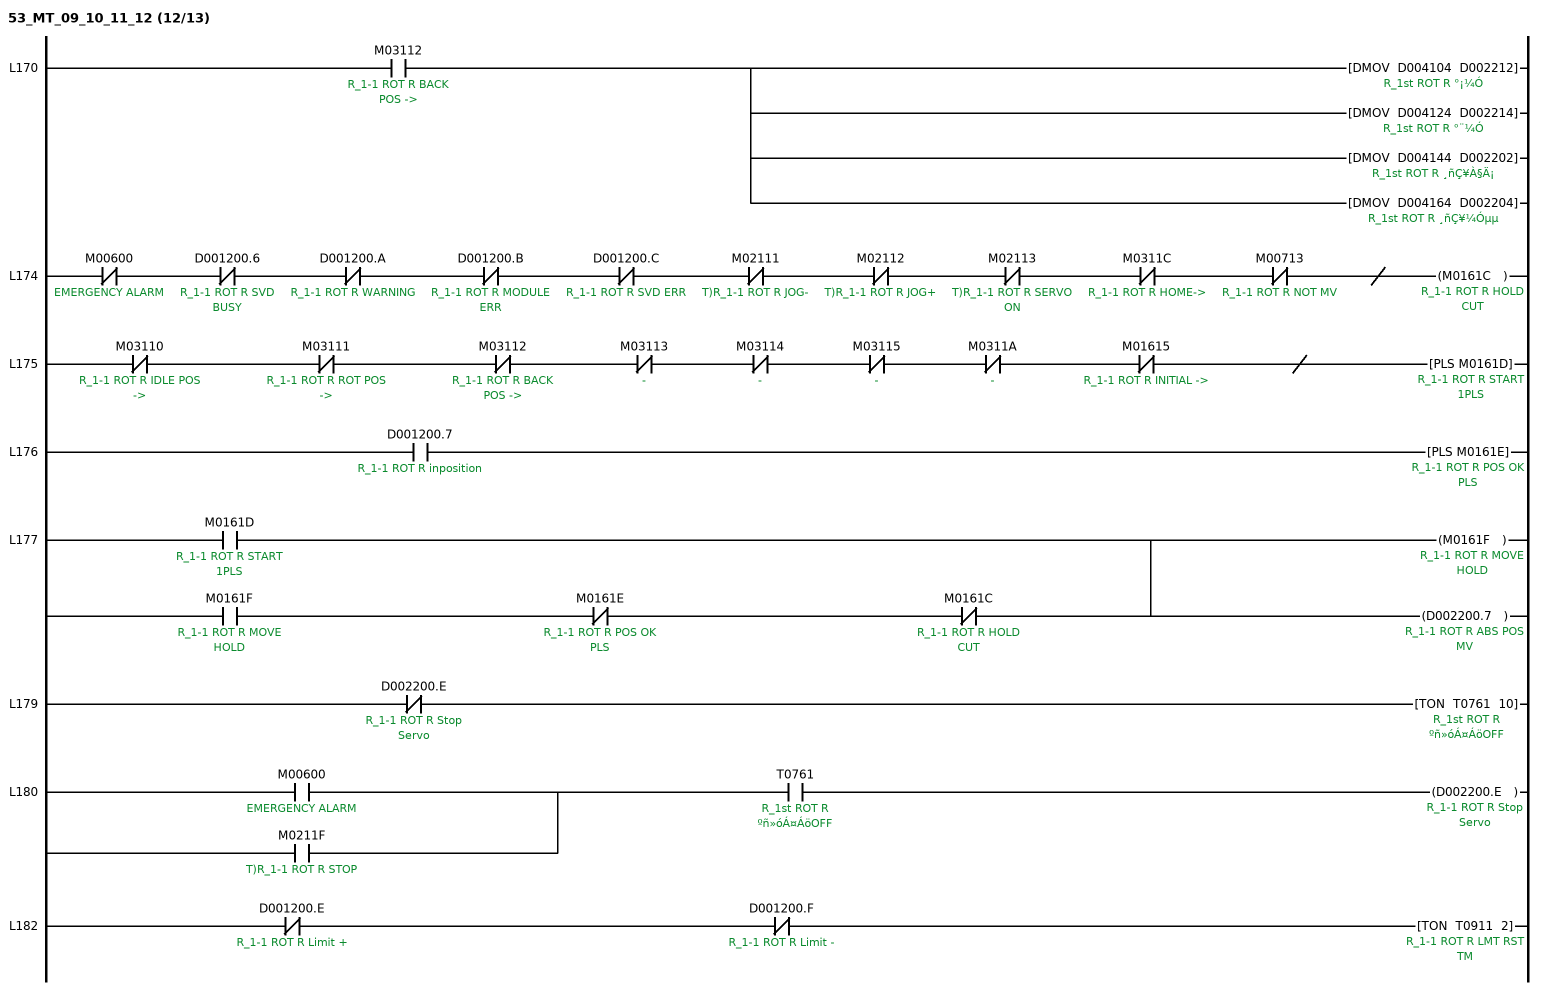
[picture p288: 53_MT_09_10_11_12 rungs L170-L182]
; L170
LOAD      M03112	// R_1-1 ROT R BACK POS ->
DMOV      D004104 D002212	// R_1st ROT R °¡¼Ó
DMOV      D004124 D002214	// R_1st ROT R °¨¼Ó
DMOV      D004144 D002202	// R_1st ROT R ¸ñÇ¥À§Ä¡
DMOV      D004164 D002204	// R_1st ROT R ¸ñÇ¥¼Óµµ
; L174
LOAD NOT  M00600	// EMERGENCY ALARM
AND NOT   D001200.6	// R_1-1 ROT R SVD BUSY
AND NOT   D001200.A	// R_1-1 ROT R WARNING
AND NOT   D001200.B	// R_1-1 ROT R MODULE ERR
AND NOT   D001200.C	// R_1-1 ROT R SVD ERR
AND NOT   M02111	// T)R_1-1 ROT R JOG-
AND NOT   M02112	// T)R_1-1 ROT R JOG+
AND NOT   M02113	// T)R_1-1 ROT R SERVO ON
AND NOT   M0311C	// R_1-1 ROT R HOME->
AND NOT   M00713	// R_1-1 ROT R NOT MV
NOT
OUT       M0161C	// R_1-1 ROT R HOLD CUT
; L175
LOAD NOT  M03110	// R_1-1 ROT R IDLE POS ->
AND NOT   M03111	// R_1-1 ROT R ROT POS ->
AND NOT   M03112	// R_1-1 ROT R BACK POS ->
AND NOT   M03113	// -
AND NOT   M03114	// -
AND NOT   M03115	// -
AND NOT   M0311A	// -
AND NOT   M01615	// R_1-1 ROT R INITIAL ->
NOT
OUTP      M0161D	// R_1-1 ROT R START 1PLS
; L176
LOAD      D001200.7	// R_1-1 ROT R inposition
OUTP      M0161E	// R_1-1 ROT R POS OK PLS
; L177
LOAD      M0161D	// R_1-1 ROT R START 1PLS
LOAD      M0161F	// R_1-1 ROT R MOVE HOLD
AND NOT   M0161E	// R_1-1 ROT R POS OK PLS
AND NOT   M0161C	// R_1-1 ROT R HOLD CUT
OR LOAD
OUT       M0161F	// R_1-1 ROT R MOVE HOLD
OUT       D002200.7	// R_1-1 ROT R ABS POS MV
; L179
LOAD NOT  D002200.E	// R_1-1 ROT R Stop Servo
TON       T0761 10	// R_1st ROT R ºñ»óÁ¤ÁöOFF
; L180
LOAD      M00600	// EMERGENCY ALARM
OR        M0211F	// T)R_1-1 ROT R STOP
AND       T0761	// R_1st ROT R ºñ»óÁ¤ÁöOFF
OUT       D002200.E	// R_1-1 ROT R Stop Servo
; L182
LOAD NOT  D001200.E	// R_1-1 ROT R Limit +
AND NOT   D001200.F	// R_1-1 ROT R Limit -
TON       T0911 2	// R_1-1 ROT R LMT RST TM

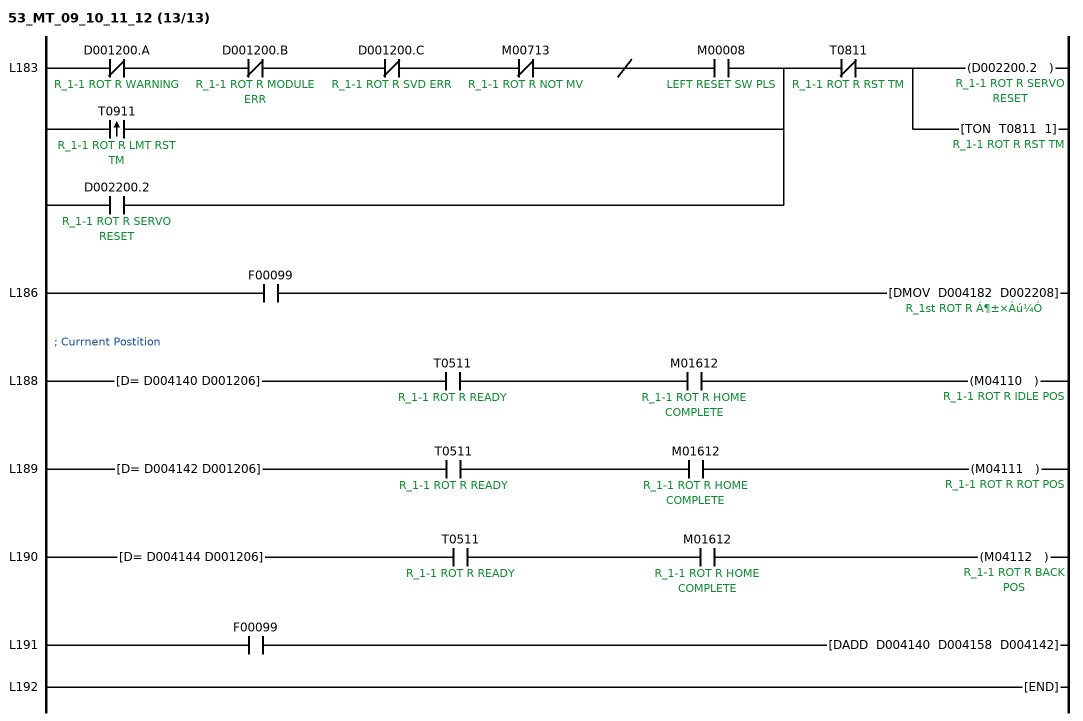
; L183
LOAD NOT  D001200.A	// R_1-1 ROT R WARNING
AND NOT   D001200.B	// R_1-1 ROT R MODULE ERR
AND NOT   D001200.C	// R_1-1 ROT R SVD ERR
AND NOT   M00713	// R_1-1 ROT R NOT MV
NOT
AND       M00008	// LEFT RESET SW PLS
ORP       T0911	// R_1-1 ROT R LMT RST TM
OR        D002200.2	// R_1-1 ROT R SERVO RESET
AND NOT   T0811	// R_1-1 ROT R RST TM
OUT       D002200.2	// R_1-1 ROT R SERVO RESET
TON       T0811 1	// R_1-1 ROT R RST TM
; L186
LOAD      F00099
DMOV      D004182 D002208	// R_1st ROT R Á¶±×Àú¼Ó
// Currnent Postition
; L188
LOADD=    D004140 D001206
AND       T0511	// R_1-1 ROT R READY
AND       M01612	// R_1-1 ROT R HOME COMPLETE
OUT       M04110	// R_1-1 ROT R IDLE POS
; L189
LOADD=    D004142 D001206
AND       T0511	// R_1-1 ROT R READY
AND       M01612	// R_1-1 ROT R HOME COMPLETE
OUT       M04111	// R_1-1 ROT R ROT POS
; L190
LOADD=    D004144 D001206
AND       T0511	// R_1-1 ROT R READY
AND       M01612	// R_1-1 ROT R HOME COMPLETE
OUT       M04112	// R_1-1 ROT R BACK POS
; L191
LOAD      F00099
DADD      D004140 D004158 D004142
; L192
END

PROGRAM 54_MT_13_14_15_16 (task: ½ºÄµ ÇÁ·Î±×·¥)

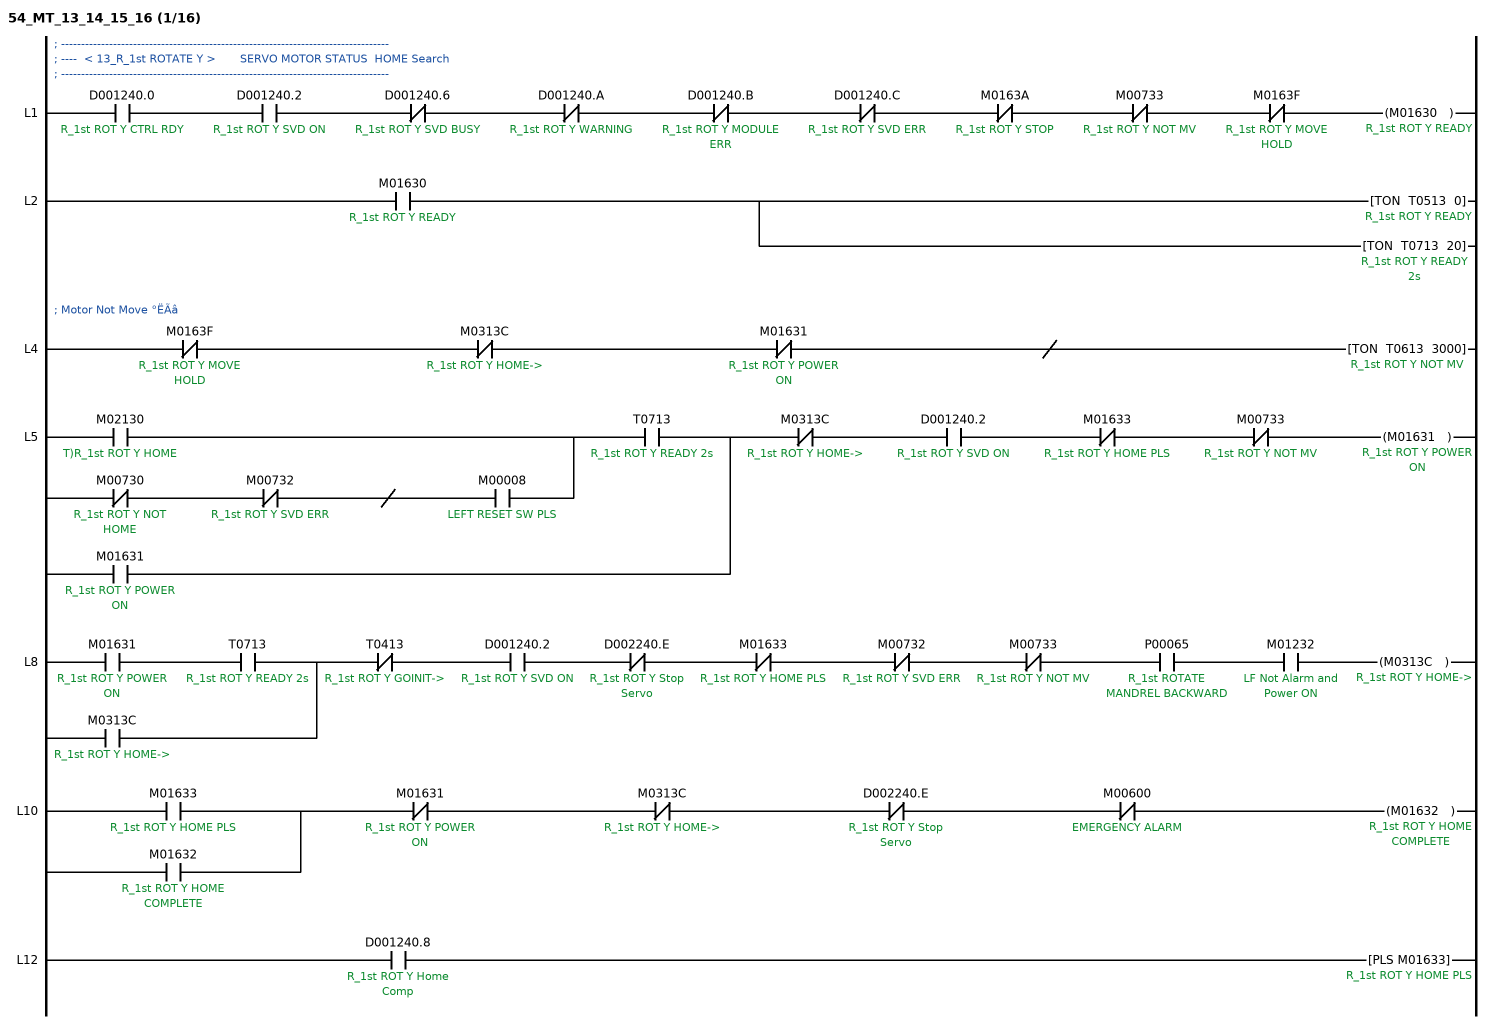
// ----------------------------------------------------------------------------------
// 
// ----  < 13_R_1st ROTATE Y >       SERVO MOTOR STATUS  HOME Search
// 
// ----------------------------------------------------------------------------------
; L1
LOAD      D001240.0	// R_1st ROT Y CTRL RDY
AND       D001240.2	// R_1st ROT Y SVD ON
AND NOT   D001240.6	// R_1st ROT Y SVD BUSY
AND NOT   D001240.A	// R_1st ROT Y WARNING
AND NOT   D001240.B	// R_1st ROT Y MODULE ERR
AND NOT   D001240.C	// R_1st ROT Y SVD ERR
AND NOT   M0163A	// R_1st ROT Y STOP
AND NOT   M00733	// R_1st ROT Y NOT MV
AND NOT   M0163F	// R_1st ROT Y MOVE HOLD
OUT       M01630	// R_1st ROT Y READY
; L2
LOAD      M01630	// R_1st ROT Y READY
TON       T0513 0	// R_1st ROT Y READY
TON       T0713 20	// R_1st ROT Y READY 2s
; L4
LOAD NOT  M0163F	// R_1st ROT Y MOVE HOLD
AND NOT   M0313C	// R_1st ROT Y HOME->
AND NOT   M01631	// R_1st ROT Y POWER ON
NOT
TON       T0613 3000	// R_1st ROT Y NOT MV
// output comment: Motor Not Move °ËÃâ
; L5
LOAD      M02130	// T)R_1st ROT Y HOME
LOAD NOT  M00730	// R_1st ROT Y NOT HOME
AND NOT   M00732	// R_1st ROT Y SVD ERR
NOT
AND       M00008	// LEFT RESET SW PLS
OR LOAD
AND       T0713	// R_1st ROT Y READY 2s
OR        M01631	// R_1st ROT Y POWER ON
AND NOT   M0313C	// R_1st ROT Y HOME->
AND       D001240.2	// R_1st ROT Y SVD ON
AND NOT   M01633	// R_1st ROT Y HOME PLS
AND NOT   M00733	// R_1st ROT Y NOT MV
OUT       M01631	// R_1st ROT Y POWER ON
; L8
LOAD      M01631	// R_1st ROT Y POWER ON
AND       T0713	// R_1st ROT Y READY 2s
OR        M0313C	// R_1st ROT Y HOME->
AND NOT   T0413	// R_1st ROT Y GOINIT->
AND       D001240.2	// R_1st ROT Y SVD ON
AND NOT   D002240.E	// R_1st ROT Y Stop Servo
AND NOT   M01633	// R_1st ROT Y HOME PLS
AND NOT   M00732	// R_1st ROT Y SVD ERR
AND NOT   M00733	// R_1st ROT Y NOT MV
AND       P00065	// R_1st ROTATE MANDREL BACKWARD
AND       M01232	// LF Not Alarm and Power ON
OUT       M0313C	// R_1st ROT Y HOME->
; L10
LOAD      M01633	// R_1st ROT Y HOME PLS
OR        M01632	// R_1st ROT Y HOME COMPLETE
AND NOT   M01631	// R_1st ROT Y POWER ON
AND NOT   M0313C	// R_1st ROT Y HOME->
AND NOT   D002240.E	// R_1st ROT Y Stop Servo
AND NOT   M00600	// EMERGENCY ALARM
OUT       M01632	// R_1st ROT Y HOME COMPLETE
; L12
LOAD      D001240.8	// R_1st ROT Y Home Comp
OUTP      M01633	// R_1st ROT Y HOME PLS

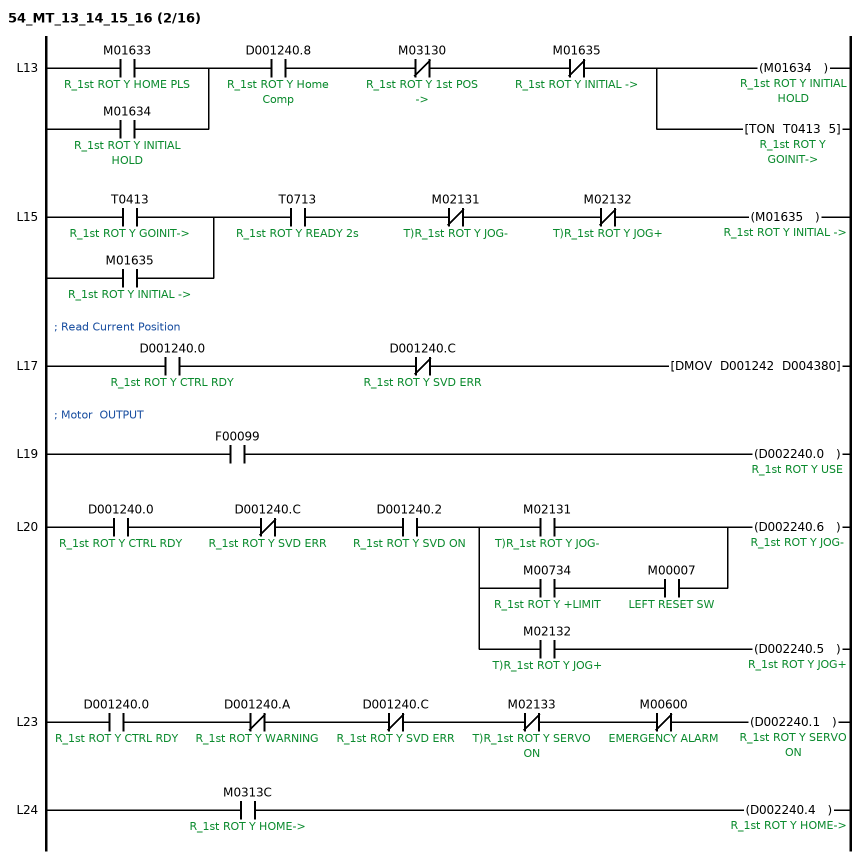
; L13
LOAD      M01633	// R_1st ROT Y HOME PLS
OR        M01634	// R_1st ROT Y INITIAL HOLD
AND       D001240.8	// R_1st ROT Y Home Comp
AND NOT   M03130	// R_1st ROT Y 1st POS ->
AND NOT   M01635	// R_1st ROT Y INITIAL ->
OUT       M01634	// R_1st ROT Y INITIAL HOLD
TON       T0413 5	// R_1st ROT Y GOINIT->
; L15
LOAD      T0413	// R_1st ROT Y GOINIT->
OR        M01635	// R_1st ROT Y INITIAL ->
AND       T0713	// R_1st ROT Y READY 2s
AND NOT   M02131	// T)R_1st ROT Y JOG-
AND NOT   M02132	// T)R_1st ROT Y JOG+
OUT       M01635	// R_1st ROT Y INITIAL ->
; L17
LOAD      D001240.0	// R_1st ROT Y CTRL RDY
AND NOT   D001240.C	// R_1st ROT Y SVD ERR
DMOV      D001242 D004380
// output comment: Read Current Position
//  Motor  OUTPUT
; L19
LOAD      F00099
OUT       D002240.0	// R_1st ROT Y USE
; L20
LOAD      D001240.0	// R_1st ROT Y CTRL RDY
AND NOT   D001240.C	// R_1st ROT Y SVD ERR
AND       D001240.2	// R_1st ROT Y SVD ON
MPUSH
LOAD      M02131	// T)R_1st ROT Y JOG-
LOAD      M00734	// R_1st ROT Y +LIMIT
AND       M00007	// LEFT RESET SW
OR LOAD
AND LOAD
OUT       D002240.6	// R_1st ROT Y JOG-
MPOP
AND       M02132	// T)R_1st ROT Y JOG+
OUT       D002240.5	// R_1st ROT Y JOG+
; L23
LOAD      D001240.0	// R_1st ROT Y CTRL RDY
AND NOT   D001240.A	// R_1st ROT Y WARNING
AND NOT   D001240.C	// R_1st ROT Y SVD ERR
AND NOT   M02133	// T)R_1st ROT Y SERVO ON
AND NOT   M00600	// EMERGENCY ALARM
OUT       D002240.1	// R_1st ROT Y SERVO ON
; L24
LOAD      M0313C	// R_1st ROT Y HOME->
OUT       D002240.4	// R_1st ROT Y HOME->

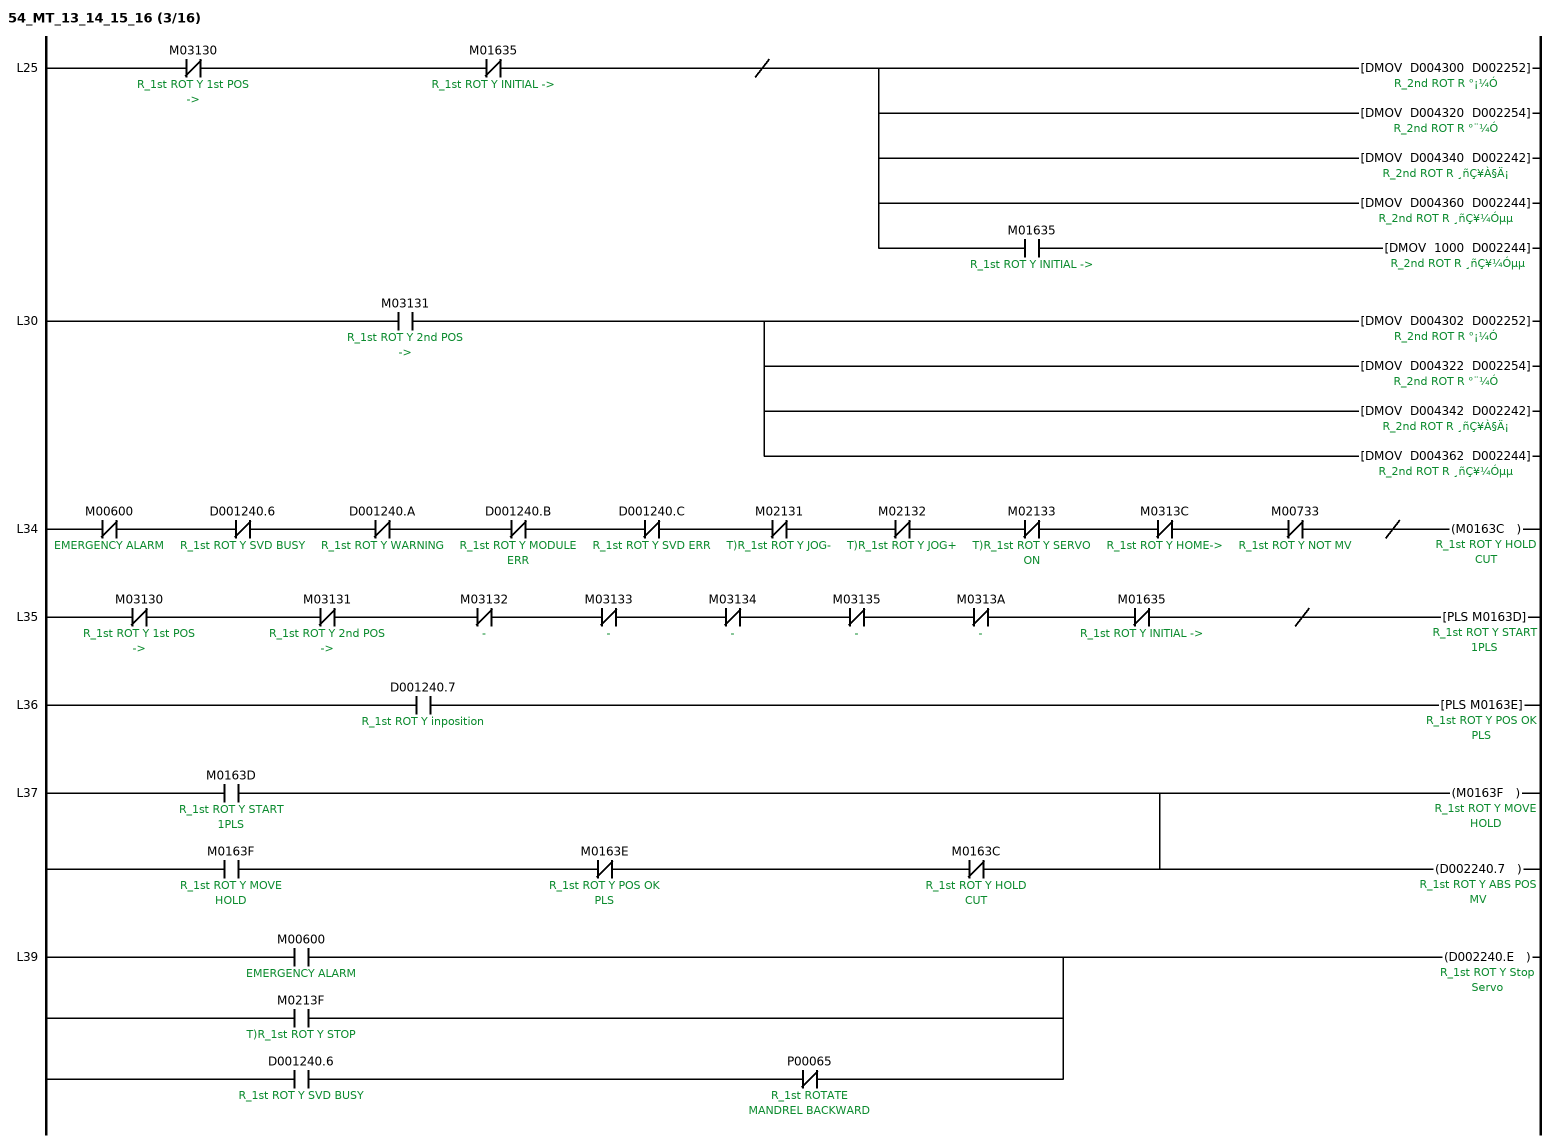
; L25
LOAD NOT  M03130	// R_1st ROT Y 1st POS ->
AND NOT   M01635	// R_1st ROT Y INITIAL ->
NOT
DMOV      D004300 D002252	// R_2nd ROT R °¡¼Ó
DMOV      D004320 D002254	// R_2nd ROT R °¨¼Ó
DMOV      D004340 D002242	// R_2nd ROT R ¸ñÇ¥À§Ä¡
DMOV      D004360 D002244	// R_2nd ROT R ¸ñÇ¥¼Óµµ
AND       M01635	// R_1st ROT Y INITIAL ->
DMOV      1000 D002244	// R_2nd ROT R ¸ñÇ¥¼Óµµ
; L30
LOAD      M03131	// R_1st ROT Y 2nd POS ->
DMOV      D004302 D002252	// R_2nd ROT R °¡¼Ó
DMOV      D004322 D002254	// R_2nd ROT R °¨¼Ó
DMOV      D004342 D002242	// R_2nd ROT R ¸ñÇ¥À§Ä¡
DMOV      D004362 D002244	// R_2nd ROT R ¸ñÇ¥¼Óµµ
; L34
LOAD NOT  M00600	// EMERGENCY ALARM
AND NOT   D001240.6	// R_1st ROT Y SVD BUSY
AND NOT   D001240.A	// R_1st ROT Y WARNING
AND NOT   D001240.B	// R_1st ROT Y MODULE ERR
AND NOT   D001240.C	// R_1st ROT Y SVD ERR
AND NOT   M02131	// T)R_1st ROT Y JOG-
AND NOT   M02132	// T)R_1st ROT Y JOG+
AND NOT   M02133	// T)R_1st ROT Y SERVO ON
AND NOT   M0313C	// R_1st ROT Y HOME->
AND NOT   M00733	// R_1st ROT Y NOT MV
NOT
OUT       M0163C	// R_1st ROT Y HOLD CUT
; L35
LOAD NOT  M03130	// R_1st ROT Y 1st POS ->
AND NOT   M03131	// R_1st ROT Y 2nd POS ->
AND NOT   M03132	// -
AND NOT   M03133	// -
AND NOT   M03134	// -
AND NOT   M03135	// -
AND NOT   M0313A	// -
AND NOT   M01635	// R_1st ROT Y INITIAL ->
NOT
OUTP      M0163D	// R_1st ROT Y START 1PLS
; L36
LOAD      D001240.7	// R_1st ROT Y inposition
OUTP      M0163E	// R_1st ROT Y POS OK PLS
; L37
LOAD      M0163D	// R_1st ROT Y START 1PLS
LOAD      M0163F	// R_1st ROT Y MOVE HOLD
AND NOT   M0163E	// R_1st ROT Y POS OK PLS
AND NOT   M0163C	// R_1st ROT Y HOLD CUT
OR LOAD
OUT       M0163F	// R_1st ROT Y MOVE HOLD
OUT       D002240.7	// R_1st ROT Y ABS POS MV
; L39
LOAD      M00600	// EMERGENCY ALARM
OR        M0213F	// T)R_1st ROT Y STOP
LOAD      D001240.6	// R_1st ROT Y SVD BUSY
AND NOT   P00065	// R_1st ROTATE MANDREL BACKWARD
OR LOAD
OUT       D002240.E	// R_1st ROT Y Stop Servo

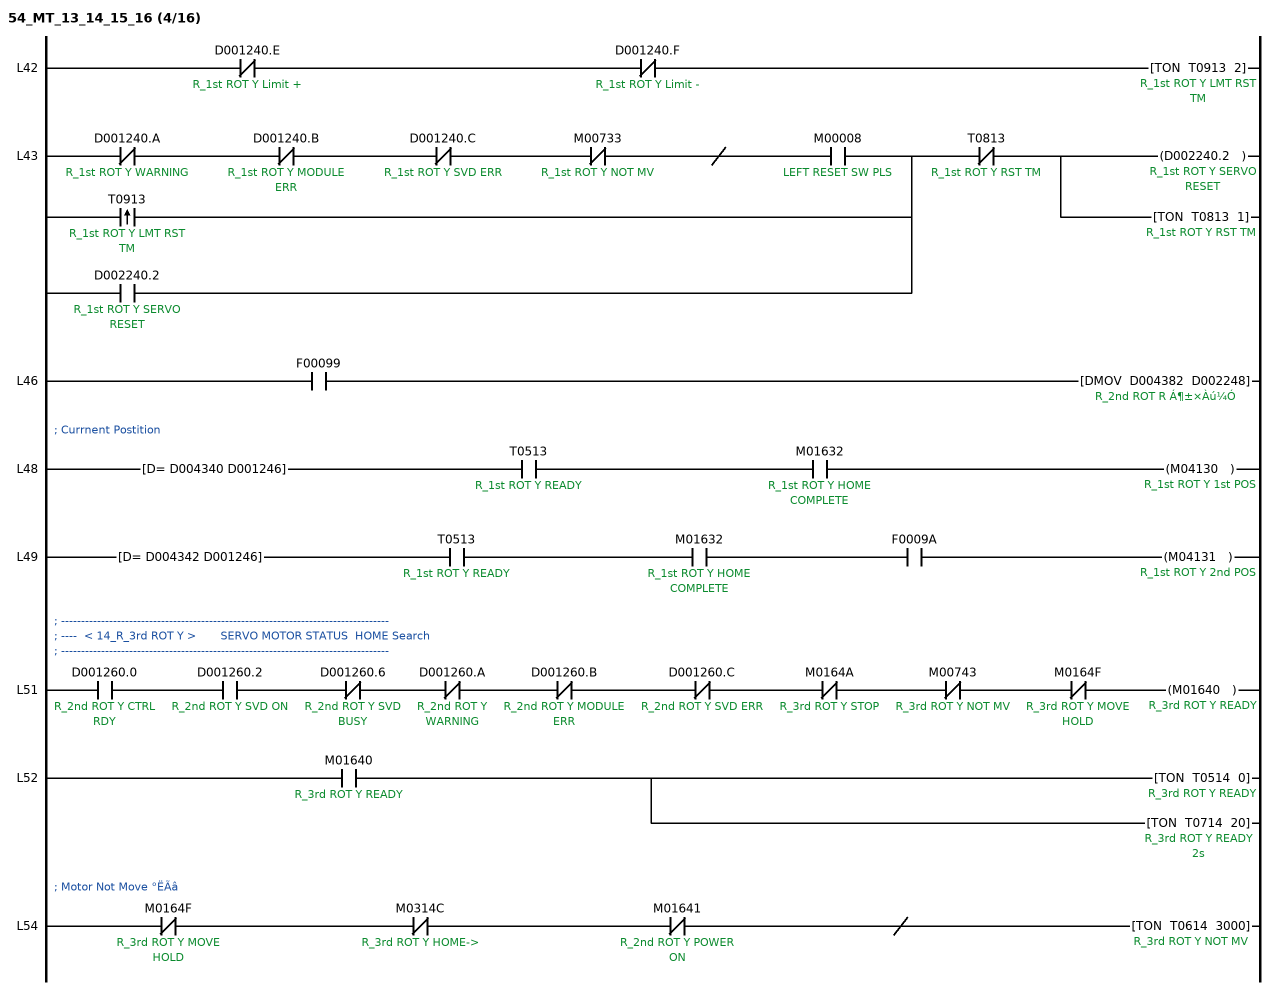
; L42
LOAD NOT  D001240.E	// R_1st ROT Y Limit +
AND NOT   D001240.F	// R_1st ROT Y Limit -
TON       T0913 2	// R_1st ROT Y LMT RST TM
; L43
LOAD NOT  D001240.A	// R_1st ROT Y WARNING
AND NOT   D001240.B	// R_1st ROT Y MODULE ERR
AND NOT   D001240.C	// R_1st ROT Y SVD ERR
AND NOT   M00733	// R_1st ROT Y NOT MV
NOT
AND       M00008	// LEFT RESET SW PLS
ORP       T0913	// R_1st ROT Y LMT RST TM
OR        D002240.2	// R_1st ROT Y SERVO RESET
AND NOT   T0813	// R_1st ROT Y RST TM
OUT       D002240.2	// R_1st ROT Y SERVO RESET
TON       T0813 1	// R_1st ROT Y RST TM
; L46
LOAD      F00099
DMOV      D004382 D002248	// R_2nd ROT R Á¶±×Àú¼Ó
// Currnent Postition
; L48
LOADD=    D004340 D001246
AND       T0513	// R_1st ROT Y READY
AND       M01632	// R_1st ROT Y HOME COMPLETE
OUT       M04130	// R_1st ROT Y 1st POS
; L49
LOADD=    D004342 D001246
AND       T0513	// R_1st ROT Y READY
AND       M01632	// R_1st ROT Y HOME COMPLETE
AND       F0009A
OUT       M04131	// R_1st ROT Y 2nd POS
// ----------------------------------------------------------------------------------
// 
// ----  < 14_R_3rd ROT Y >       SERVO MOTOR STATUS  HOME Search
// 
// ----------------------------------------------------------------------------------
; L51
LOAD      D001260.0	// R_2nd ROT Y CTRL RDY
AND       D001260.2	// R_2nd ROT Y SVD ON
AND NOT   D001260.6	// R_2nd ROT Y SVD BUSY
AND NOT   D001260.A	// R_2nd ROT Y WARNING
AND NOT   D001260.B	// R_2nd ROT Y MODULE ERR
AND NOT   D001260.C	// R_2nd ROT Y SVD ERR
AND NOT   M0164A	// R_3rd ROT Y STOP
AND NOT   M00743	// R_3rd ROT Y NOT MV
AND NOT   M0164F	// R_3rd ROT Y MOVE HOLD
OUT       M01640	// R_3rd ROT Y READY
; L52
LOAD      M01640	// R_3rd ROT Y READY
TON       T0514 0	// R_3rd ROT Y READY
TON       T0714 20	// R_3rd ROT Y READY 2s
; L54
LOAD NOT  M0164F	// R_3rd ROT Y MOVE HOLD
AND NOT   M0314C	// R_3rd ROT Y HOME->
AND NOT   M01641	// R_2nd ROT Y POWER ON
NOT
TON       T0614 3000	// R_3rd ROT Y NOT MV
// output comment: Motor Not Move °ËÃâ

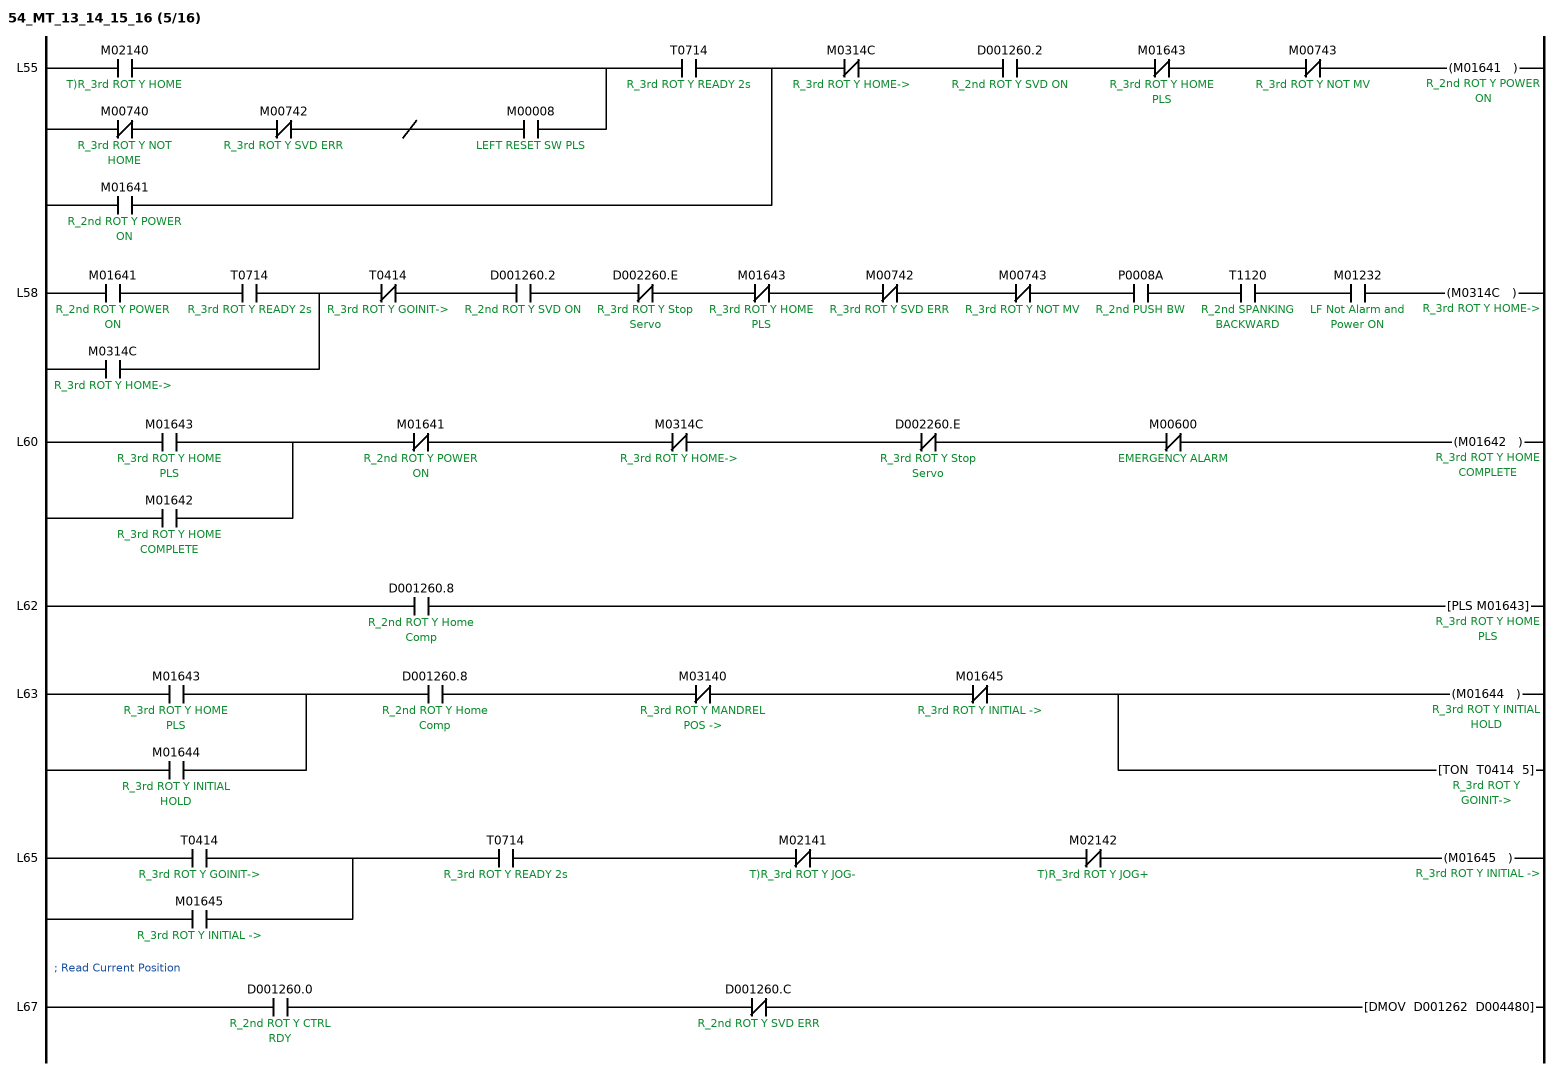
; L55
LOAD      M02140	// T)R_3rd ROT Y HOME
LOAD NOT  M00740	// R_3rd ROT Y NOT HOME
AND NOT   M00742	// R_3rd ROT Y SVD ERR
NOT
AND       M00008	// LEFT RESET SW PLS
OR LOAD
AND       T0714	// R_3rd ROT Y READY 2s
OR        M01641	// R_2nd ROT Y POWER ON
AND NOT   M0314C	// R_3rd ROT Y HOME->
AND       D001260.2	// R_2nd ROT Y SVD ON
AND NOT   M01643	// R_3rd ROT Y HOME PLS
AND NOT   M00743	// R_3rd ROT Y NOT MV
OUT       M01641	// R_2nd ROT Y POWER ON
; L58
LOAD      M01641	// R_2nd ROT Y POWER ON
AND       T0714	// R_3rd ROT Y READY 2s
OR        M0314C	// R_3rd ROT Y HOME->
AND NOT   T0414	// R_3rd ROT Y GOINIT->
AND       D001260.2	// R_2nd ROT Y SVD ON
AND NOT   D002260.E	// R_3rd ROT Y Stop Servo
AND NOT   M01643	// R_3rd ROT Y HOME PLS
AND NOT   M00742	// R_3rd ROT Y SVD ERR
AND NOT   M00743	// R_3rd ROT Y NOT MV
AND       P0008A	// R_2nd PUSH BW
AND       T1120	// R_2nd SPANKING BACKWARD
AND       M01232	// LF Not Alarm and Power ON
OUT       M0314C	// R_3rd ROT Y HOME->
; L60
LOAD      M01643	// R_3rd ROT Y HOME PLS
OR        M01642	// R_3rd ROT Y HOME COMPLETE
AND NOT   M01641	// R_2nd ROT Y POWER ON
AND NOT   M0314C	// R_3rd ROT Y HOME->
AND NOT   D002260.E	// R_3rd ROT Y Stop Servo
AND NOT   M00600	// EMERGENCY ALARM
OUT       M01642	// R_3rd ROT Y HOME COMPLETE
; L62
LOAD      D001260.8	// R_2nd ROT Y Home Comp
OUTP      M01643	// R_3rd ROT Y HOME PLS
; L63
LOAD      M01643	// R_3rd ROT Y HOME PLS
OR        M01644	// R_3rd ROT Y INITIAL HOLD
AND       D001260.8	// R_2nd ROT Y Home Comp
AND NOT   M03140	// R_3rd ROT Y MANDREL POS ->
AND NOT   M01645	// R_3rd ROT Y INITIAL ->
OUT       M01644	// R_3rd ROT Y INITIAL HOLD
TON       T0414 5	// R_3rd ROT Y GOINIT->
; L65
LOAD      T0414	// R_3rd ROT Y GOINIT->
OR        M01645	// R_3rd ROT Y INITIAL ->
AND       T0714	// R_3rd ROT Y READY 2s
AND NOT   M02141	// T)R_3rd ROT Y JOG-
AND NOT   M02142	// T)R_3rd ROT Y JOG+
OUT       M01645	// R_3rd ROT Y INITIAL ->
; L67
LOAD      D001260.0	// R_2nd ROT Y CTRL RDY
AND NOT   D001260.C	// R_2nd ROT Y SVD ERR
DMOV      D001262 D004480
// output comment: Read Current Position

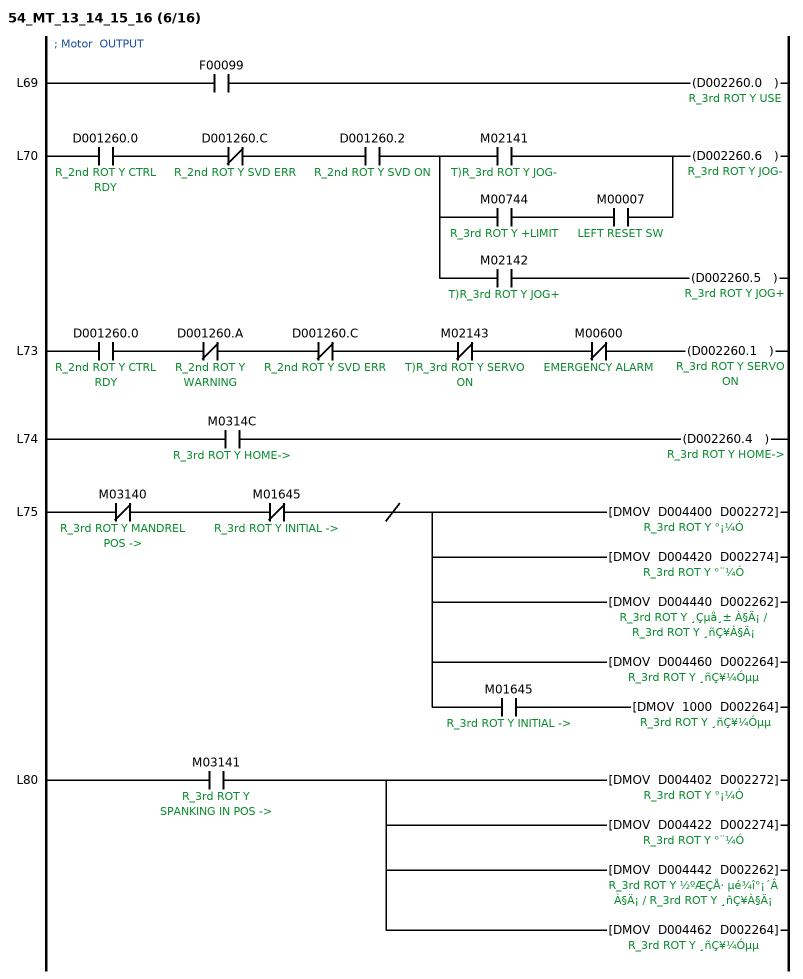
//  Motor  OUTPUT
; L69
LOAD      F00099
OUT       D002260.0	// R_3rd ROT Y USE
; L70
LOAD      D001260.0	// R_2nd ROT Y CTRL RDY
AND NOT   D001260.C	// R_2nd ROT Y SVD ERR
AND       D001260.2	// R_2nd ROT Y SVD ON
MPUSH
LOAD      M02141	// T)R_3rd ROT Y JOG-
LOAD      M00744	// R_3rd ROT Y +LIMIT
AND       M00007	// LEFT RESET SW
OR LOAD
AND LOAD
OUT       D002260.6	// R_3rd ROT Y JOG-
MPOP
AND       M02142	// T)R_3rd ROT Y JOG+
OUT       D002260.5	// R_3rd ROT Y JOG+
; L73
LOAD      D001260.0	// R_2nd ROT Y CTRL RDY
AND NOT   D001260.A	// R_2nd ROT Y WARNING
AND NOT   D001260.C	// R_2nd ROT Y SVD ERR
AND NOT   M02143	// T)R_3rd ROT Y SERVO ON
AND NOT   M00600	// EMERGENCY ALARM
OUT       D002260.1	// R_3rd ROT Y SERVO ON
; L74
LOAD      M0314C	// R_3rd ROT Y HOME->
OUT       D002260.4	// R_3rd ROT Y HOME->
; L75
LOAD NOT  M03140	// R_3rd ROT Y MANDREL POS ->
AND NOT   M01645	// R_3rd ROT Y INITIAL ->
NOT
DMOV      D004400 D002272	// R_3rd ROT Y °¡¼Ó
DMOV      D004420 D002274	// R_3rd ROT Y °¨¼Ó
DMOV      D004440 D002262	// R_3rd ROT Y ¸Çµå¸± À§Ä¡ / R_3rd ROT Y ¸ñÇ¥À§Ä¡
DMOV      D004460 D002264	// R_3rd ROT Y ¸ñÇ¥¼Óµµ
AND       M01645	// R_3rd ROT Y INITIAL ->
DMOV      1000 D002264	// R_3rd ROT Y ¸ñÇ¥¼Óµµ
; L80
LOAD      M03141	// R_3rd ROT Y SPANKING IN POS ->
DMOV      D004402 D002272	// R_3rd ROT Y °¡¼Ó
DMOV      D004422 D002274	// R_3rd ROT Y °¨¼Ó
DMOV      D004442 D002262	// R_3rd ROT Y ½ºÆÇÅ· µé¾î°¡´Â À§Ä¡ / R_3rd ROT Y ¸ñÇ¥À§Ä¡
DMOV      D004462 D002264	// R_3rd ROT Y ¸ñÇ¥¼Óµµ

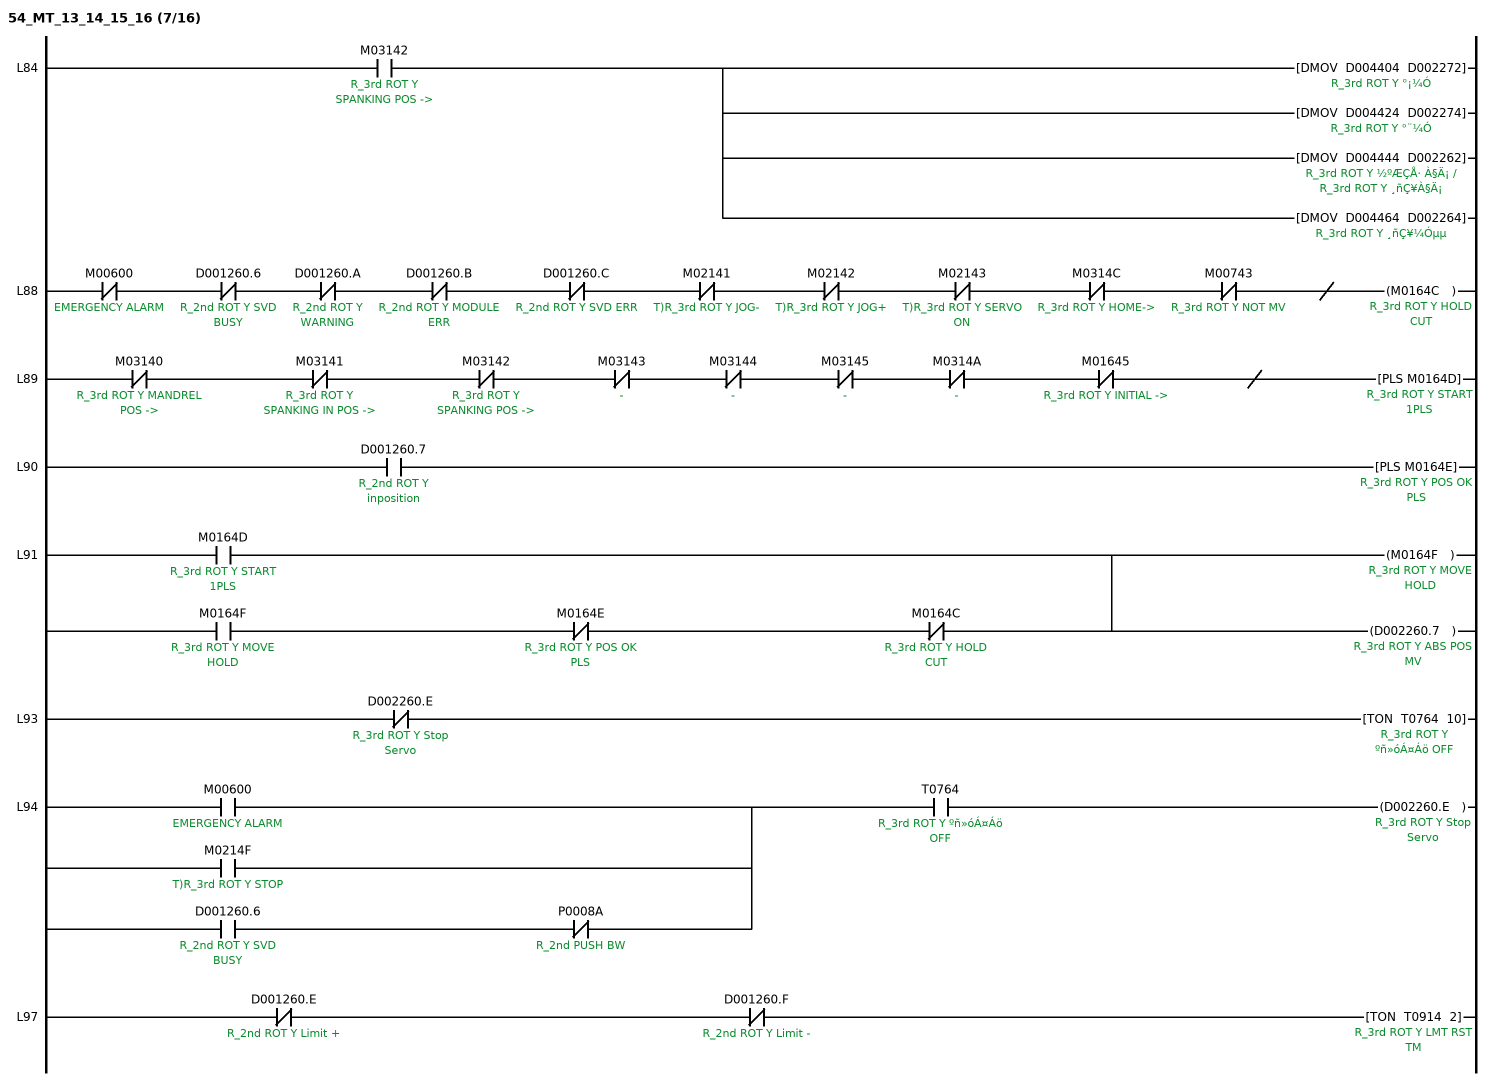
; L84
LOAD      M03142	// R_3rd ROT Y SPANKING POS ->
DMOV      D004404 D002272	// R_3rd ROT Y °¡¼Ó
DMOV      D004424 D002274	// R_3rd ROT Y °¨¼Ó
DMOV      D004444 D002262	// R_3rd ROT Y ½ºÆÇÅ· À§Ä¡ / R_3rd ROT Y ¸ñÇ¥À§Ä¡
DMOV      D004464 D002264	// R_3rd ROT Y ¸ñÇ¥¼Óµµ
; L88
LOAD NOT  M00600	// EMERGENCY ALARM
AND NOT   D001260.6	// R_2nd ROT Y SVD BUSY
AND NOT   D001260.A	// R_2nd ROT Y WARNING
AND NOT   D001260.B	// R_2nd ROT Y MODULE ERR
AND NOT   D001260.C	// R_2nd ROT Y SVD ERR
AND NOT   M02141	// T)R_3rd ROT Y JOG-
AND NOT   M02142	// T)R_3rd ROT Y JOG+
AND NOT   M02143	// T)R_3rd ROT Y SERVO ON
AND NOT   M0314C	// R_3rd ROT Y HOME->
AND NOT   M00743	// R_3rd ROT Y NOT MV
NOT
OUT       M0164C	// R_3rd ROT Y HOLD CUT
; L89
LOAD NOT  M03140	// R_3rd ROT Y MANDREL POS ->
AND NOT   M03141	// R_3rd ROT Y SPANKING IN POS ->
AND NOT   M03142	// R_3rd ROT Y SPANKING POS ->
AND NOT   M03143	// -
AND NOT   M03144	// -
AND NOT   M03145	// -
AND NOT   M0314A	// -
AND NOT   M01645	// R_3rd ROT Y INITIAL ->
NOT
OUTP      M0164D	// R_3rd ROT Y START 1PLS
; L90
LOAD      D001260.7	// R_2nd ROT Y inposition
OUTP      M0164E	// R_3rd ROT Y POS OK PLS
; L91
LOAD      M0164D	// R_3rd ROT Y START 1PLS
LOAD      M0164F	// R_3rd ROT Y MOVE HOLD
AND NOT   M0164E	// R_3rd ROT Y POS OK PLS
AND NOT   M0164C	// R_3rd ROT Y HOLD CUT
OR LOAD
OUT       M0164F	// R_3rd ROT Y MOVE HOLD
OUT       D002260.7	// R_3rd ROT Y ABS POS MV
; L93
LOAD NOT  D002260.E	// R_3rd ROT Y Stop Servo
TON       T0764 10	// R_3rd ROT Y ºñ»óÁ¤Áö OFF
; L94
LOAD      M00600	// EMERGENCY ALARM
OR        M0214F	// T)R_3rd ROT Y STOP
LOAD      D001260.6	// R_2nd ROT Y SVD BUSY
AND NOT   P0008A	// R_2nd PUSH BW
OR LOAD
AND       T0764	// R_3rd ROT Y ºñ»óÁ¤Áö OFF
OUT       D002260.E	// R_3rd ROT Y Stop Servo
; L97
LOAD NOT  D001260.E	// R_2nd ROT Y Limit +
AND NOT   D001260.F	// R_2nd ROT Y Limit -
TON       T0914 2	// R_3rd ROT Y LMT RST TM

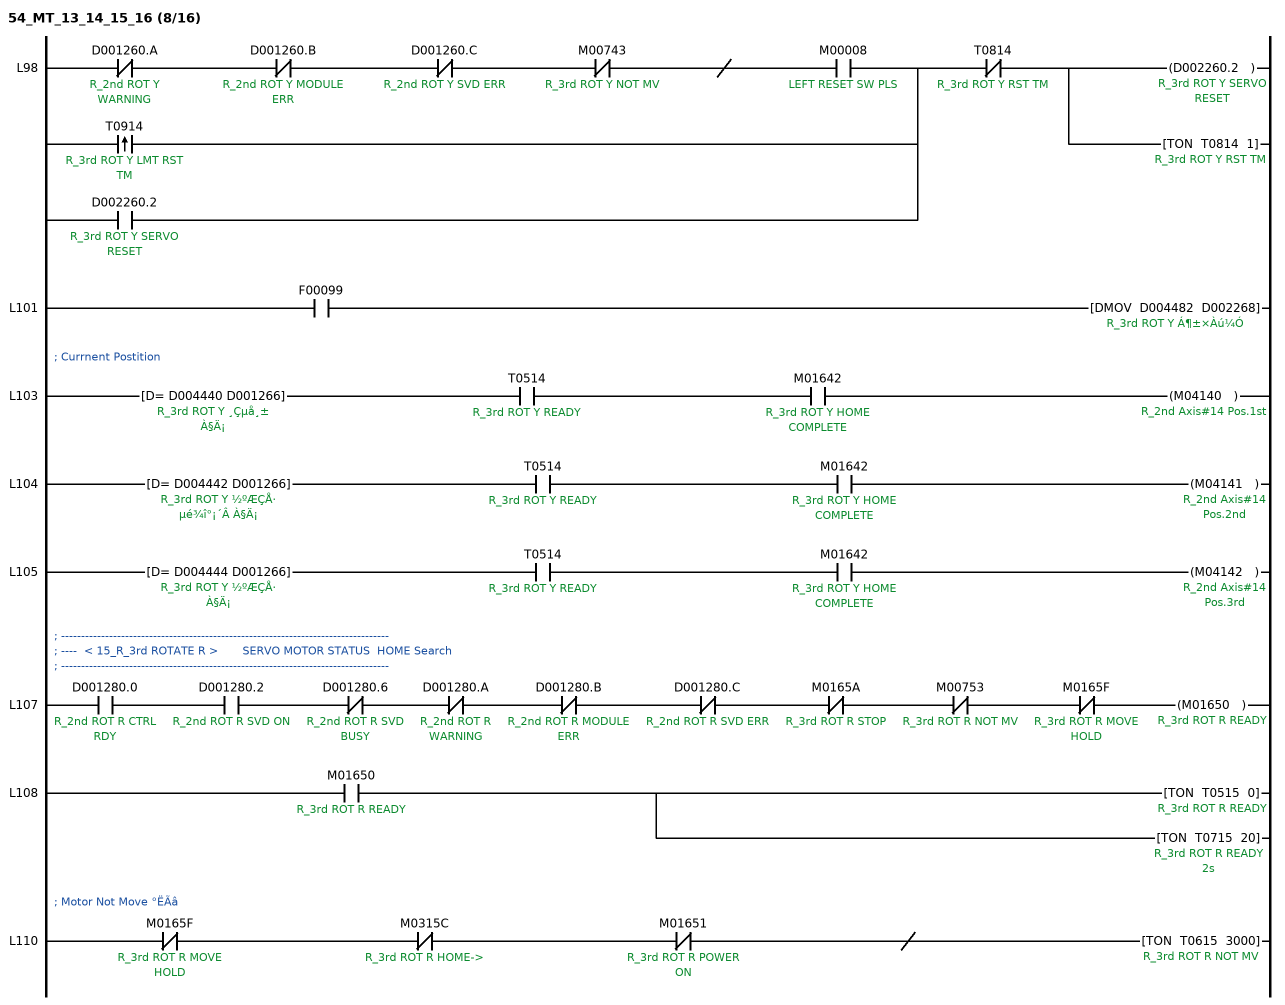
; L98
LOAD NOT  D001260.A	// R_2nd ROT Y WARNING
AND NOT   D001260.B	// R_2nd ROT Y MODULE ERR
AND NOT   D001260.C	// R_2nd ROT Y SVD ERR
AND NOT   M00743	// R_3rd ROT Y NOT MV
NOT
AND       M00008	// LEFT RESET SW PLS
ORP       T0914	// R_3rd ROT Y LMT RST TM
OR        D002260.2	// R_3rd ROT Y SERVO RESET
AND NOT   T0814	// R_3rd ROT Y RST TM
OUT       D002260.2	// R_3rd ROT Y SERVO RESET
TON       T0814 1	// R_3rd ROT Y RST TM
; L101
LOAD      F00099
DMOV      D004482 D002268	// R_3rd ROT Y Á¶±×Àú¼Ó
// Currnent Postition
; L103
LOADD=    D004440 D001266	// R_3rd ROT Y ¸Çµå¸± À§Ä¡
AND       T0514	// R_3rd ROT Y READY
AND       M01642	// R_3rd ROT Y HOME COMPLETE
OUT       M04140	// R_2nd Axis#14 Pos.1st
; L104
LOADD=    D004442 D001266	// R_3rd ROT Y ½ºÆÇÅ· µé¾î°¡´Â À§Ä¡
AND       T0514	// R_3rd ROT Y READY
AND       M01642	// R_3rd ROT Y HOME COMPLETE
OUT       M04141	// R_2nd Axis#14 Pos.2nd
; L105
LOADD=    D004444 D001266	// R_3rd ROT Y ½ºÆÇÅ· À§Ä¡
AND       T0514	// R_3rd ROT Y READY
AND       M01642	// R_3rd ROT Y HOME COMPLETE
OUT       M04142	// R_2nd Axis#14 Pos.3rd
// ----------------------------------------------------------------------------------
// 
// ----  < 15_R_3rd ROTATE R >       SERVO MOTOR STATUS  HOME Search
// 
// ----------------------------------------------------------------------------------
; L107
LOAD      D001280.0	// R_2nd ROT R CTRL RDY
AND       D001280.2	// R_2nd ROT R SVD ON
AND NOT   D001280.6	// R_2nd ROT R SVD BUSY
AND NOT   D001280.A	// R_2nd ROT R WARNING
AND NOT   D001280.B	// R_2nd ROT R MODULE ERR
AND NOT   D001280.C	// R_2nd ROT R SVD ERR
AND NOT   M0165A	// R_3rd ROT R STOP
AND NOT   M00753	// R_3rd ROT R NOT MV
AND NOT   M0165F	// R_3rd ROT R MOVE HOLD
OUT       M01650	// R_3rd ROT R READY
; L108
LOAD      M01650	// R_3rd ROT R READY
TON       T0515 0	// R_3rd ROT R READY
TON       T0715 20	// R_3rd ROT R READY 2s
; L110
LOAD NOT  M0165F	// R_3rd ROT R MOVE HOLD
AND NOT   M0315C	// R_3rd ROT R HOME->
AND NOT   M01651	// R_3rd ROT R POWER ON
NOT
TON       T0615 3000	// R_3rd ROT R NOT MV
// output comment: Motor Not Move °ËÃâ

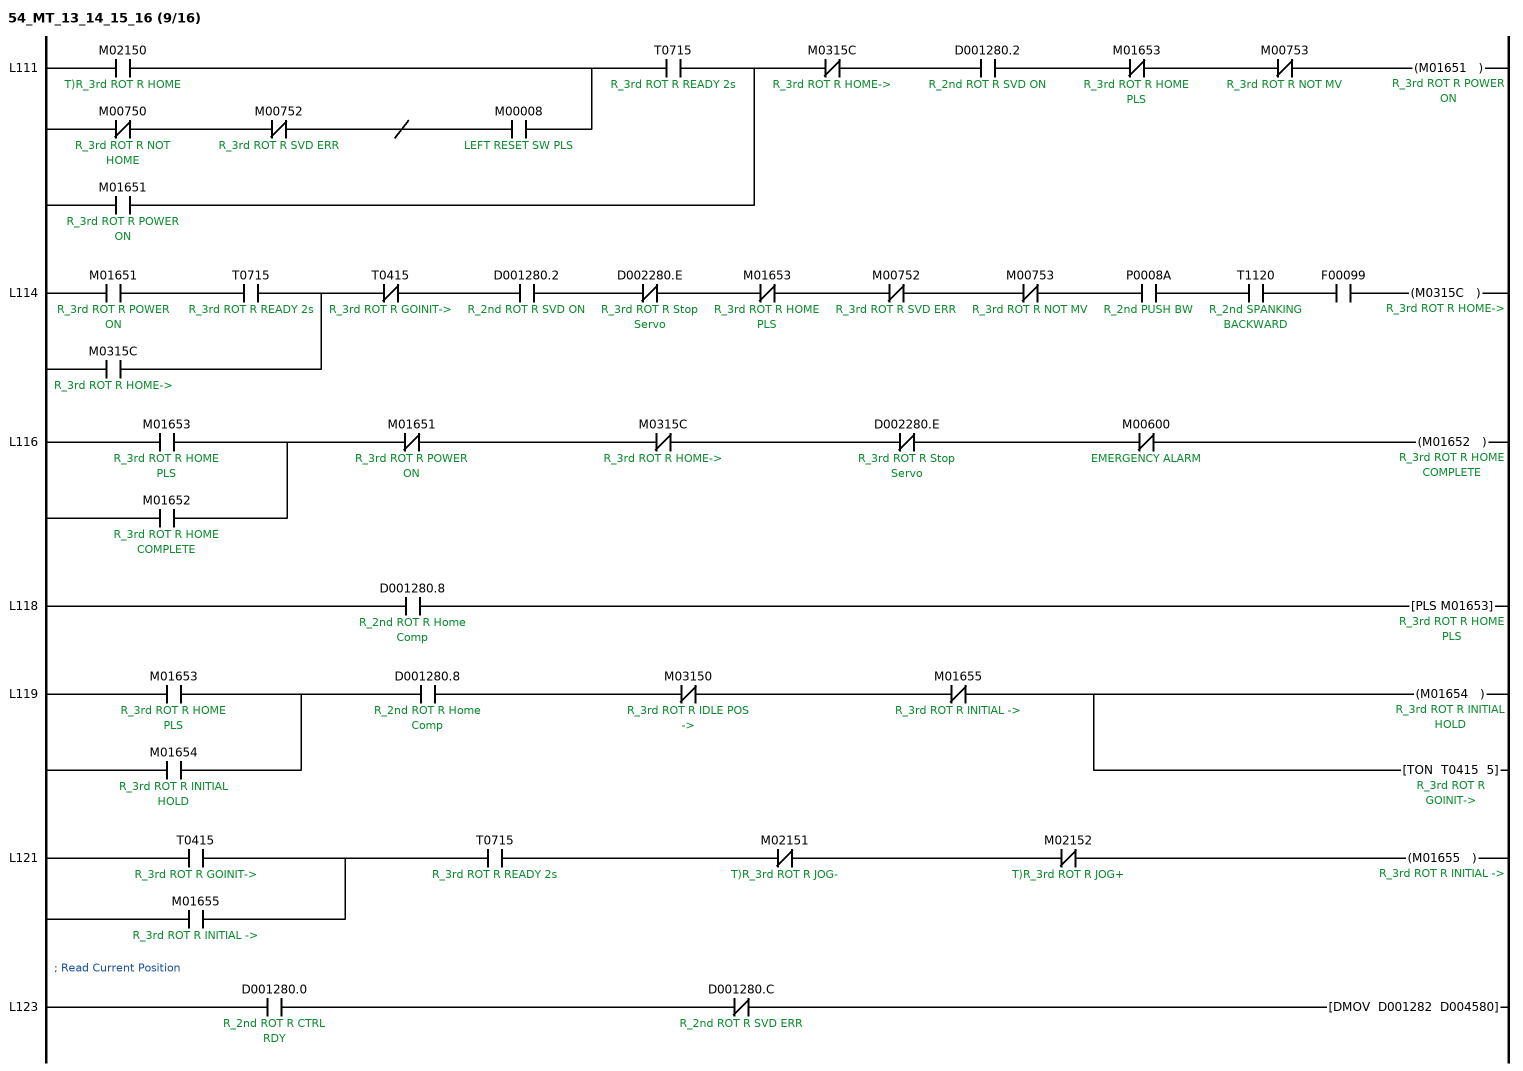
; L111
LOAD      M02150	// T)R_3rd ROT R HOME
LOAD NOT  M00750	// R_3rd ROT R NOT HOME
AND NOT   M00752	// R_3rd ROT R SVD ERR
NOT
AND       M00008	// LEFT RESET SW PLS
OR LOAD
AND       T0715	// R_3rd ROT R READY 2s
OR        M01651	// R_3rd ROT R POWER ON
AND NOT   M0315C	// R_3rd ROT R HOME->
AND       D001280.2	// R_2nd ROT R SVD ON
AND NOT   M01653	// R_3rd ROT R HOME PLS
AND NOT   M00753	// R_3rd ROT R NOT MV
OUT       M01651	// R_3rd ROT R POWER ON
; L114
LOAD      M01651	// R_3rd ROT R POWER ON
AND       T0715	// R_3rd ROT R READY 2s
OR        M0315C	// R_3rd ROT R HOME->
AND NOT   T0415	// R_3rd ROT R GOINIT->
AND       D001280.2	// R_2nd ROT R SVD ON
AND NOT   D002280.E	// R_3rd ROT R Stop Servo
AND NOT   M01653	// R_3rd ROT R HOME PLS
AND NOT   M00752	// R_3rd ROT R SVD ERR
AND NOT   M00753	// R_3rd ROT R NOT MV
AND       P0008A	// R_2nd PUSH BW
AND       T1120	// R_2nd SPANKING BACKWARD
AND       F00099
OUT       M0315C	// R_3rd ROT R HOME->
; L116
LOAD      M01653	// R_3rd ROT R HOME PLS
OR        M01652	// R_3rd ROT R HOME COMPLETE
AND NOT   M01651	// R_3rd ROT R POWER ON
AND NOT   M0315C	// R_3rd ROT R HOME->
AND NOT   D002280.E	// R_3rd ROT R Stop Servo
AND NOT   M00600	// EMERGENCY ALARM
OUT       M01652	// R_3rd ROT R HOME COMPLETE
; L118
LOAD      D001280.8	// R_2nd ROT R Home Comp
OUTP      M01653	// R_3rd ROT R HOME PLS
; L119
LOAD      M01653	// R_3rd ROT R HOME PLS
OR        M01654	// R_3rd ROT R INITIAL HOLD
AND       D001280.8	// R_2nd ROT R Home Comp
AND NOT   M03150	// R_3rd ROT R IDLE POS ->
AND NOT   M01655	// R_3rd ROT R INITIAL ->
OUT       M01654	// R_3rd ROT R INITIAL HOLD
TON       T0415 5	// R_3rd ROT R GOINIT->
; L121
LOAD      T0415	// R_3rd ROT R GOINIT->
OR        M01655	// R_3rd ROT R INITIAL ->
AND       T0715	// R_3rd ROT R READY 2s
AND NOT   M02151	// T)R_3rd ROT R JOG-
AND NOT   M02152	// T)R_3rd ROT R JOG+
OUT       M01655	// R_3rd ROT R INITIAL ->
; L123
LOAD      D001280.0	// R_2nd ROT R CTRL RDY
AND NOT   D001280.C	// R_2nd ROT R SVD ERR
DMOV      D001282 D004580
// output comment: Read Current Position

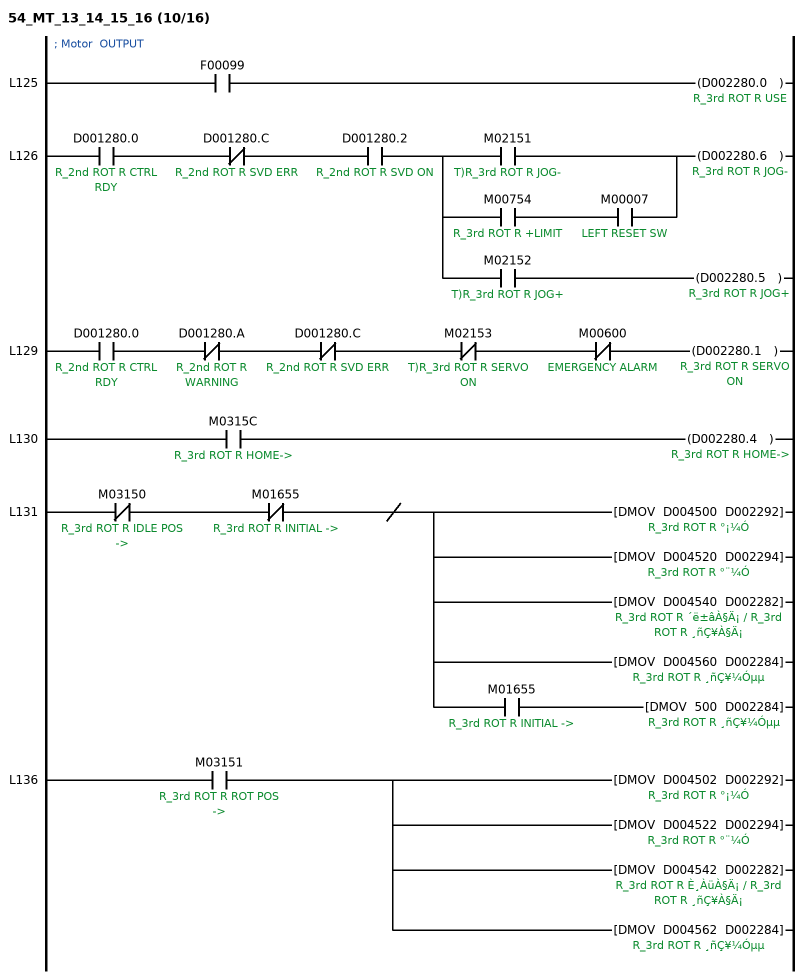
//  Motor  OUTPUT
; L125
LOAD      F00099
OUT       D002280.0	// R_3rd ROT R USE
; L126
LOAD      D001280.0	// R_2nd ROT R CTRL RDY
AND NOT   D001280.C	// R_2nd ROT R SVD ERR
AND       D001280.2	// R_2nd ROT R SVD ON
MPUSH
LOAD      M02151	// T)R_3rd ROT R JOG-
LOAD      M00754	// R_3rd ROT R +LIMIT
AND       M00007	// LEFT RESET SW
OR LOAD
AND LOAD
OUT       D002280.6	// R_3rd ROT R JOG-
MPOP
AND       M02152	// T)R_3rd ROT R JOG+
OUT       D002280.5	// R_3rd ROT R JOG+
; L129
LOAD      D001280.0	// R_2nd ROT R CTRL RDY
AND NOT   D001280.A	// R_2nd ROT R WARNING
AND NOT   D001280.C	// R_2nd ROT R SVD ERR
AND NOT   M02153	// T)R_3rd ROT R SERVO ON
AND NOT   M00600	// EMERGENCY ALARM
OUT       D002280.1	// R_3rd ROT R SERVO ON
; L130
LOAD      M0315C	// R_3rd ROT R HOME->
OUT       D002280.4	// R_3rd ROT R HOME->
; L131
LOAD NOT  M03150	// R_3rd ROT R IDLE POS ->
AND NOT   M01655	// R_3rd ROT R INITIAL ->
NOT
DMOV      D004500 D002292	// R_3rd ROT R °¡¼Ó
DMOV      D004520 D002294	// R_3rd ROT R °¨¼Ó
DMOV      D004540 D002282	// R_3rd ROT R ´ë±âÀ§Ä¡ / R_3rd ROT R ¸ñÇ¥À§Ä¡
DMOV      D004560 D002284	// R_3rd ROT R ¸ñÇ¥¼Óµµ
AND       M01655	// R_3rd ROT R INITIAL ->
DMOV      500 D002284	// R_3rd ROT R ¸ñÇ¥¼Óµµ
; L136
LOAD      M03151	// R_3rd ROT R ROT POS ->
DMOV      D004502 D002292	// R_3rd ROT R °¡¼Ó
DMOV      D004522 D002294	// R_3rd ROT R °¨¼Ó
DMOV      D004542 D002282	// R_3rd ROT R È¸ÀüÀ§Ä¡ / R_3rd ROT R ¸ñÇ¥À§Ä¡
DMOV      D004562 D002284	// R_3rd ROT R ¸ñÇ¥¼Óµµ

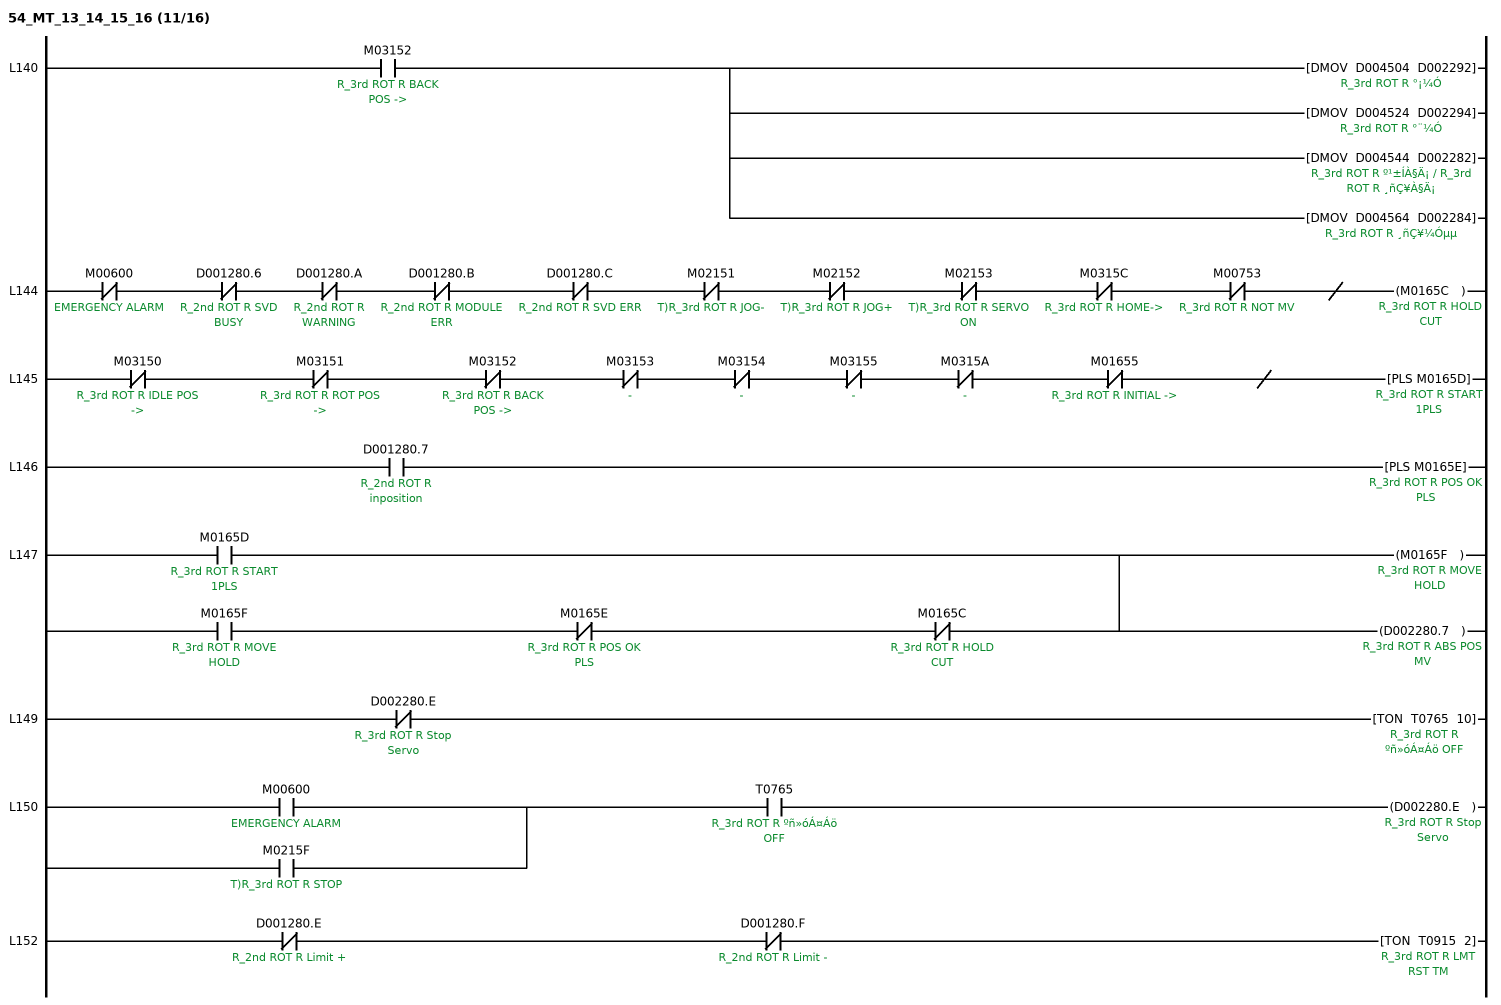
; L140
LOAD      M03152	// R_3rd ROT R BACK POS ->
DMOV      D004504 D002292	// R_3rd ROT R °¡¼Ó
DMOV      D004524 D002294	// R_3rd ROT R °¨¼Ó
DMOV      D004544 D002282	// R_3rd ROT R º¹±ÍÀ§Ä¡ / R_3rd ROT R ¸ñÇ¥À§Ä¡
DMOV      D004564 D002284	// R_3rd ROT R ¸ñÇ¥¼Óµµ
; L144
LOAD NOT  M00600	// EMERGENCY ALARM
AND NOT   D001280.6	// R_2nd ROT R SVD BUSY
AND NOT   D001280.A	// R_2nd ROT R WARNING
AND NOT   D001280.B	// R_2nd ROT R MODULE ERR
AND NOT   D001280.C	// R_2nd ROT R SVD ERR
AND NOT   M02151	// T)R_3rd ROT R JOG-
AND NOT   M02152	// T)R_3rd ROT R JOG+
AND NOT   M02153	// T)R_3rd ROT R SERVO ON
AND NOT   M0315C	// R_3rd ROT R HOME->
AND NOT   M00753	// R_3rd ROT R NOT MV
NOT
OUT       M0165C	// R_3rd ROT R HOLD CUT
; L145
LOAD NOT  M03150	// R_3rd ROT R IDLE POS ->
AND NOT   M03151	// R_3rd ROT R ROT POS ->
AND NOT   M03152	// R_3rd ROT R BACK POS ->
AND NOT   M03153	// -
AND NOT   M03154	// -
AND NOT   M03155	// -
AND NOT   M0315A	// -
AND NOT   M01655	// R_3rd ROT R INITIAL ->
NOT
OUTP      M0165D	// R_3rd ROT R START 1PLS
; L146
LOAD      D001280.7	// R_2nd ROT R inposition
OUTP      M0165E	// R_3rd ROT R POS OK PLS
; L147
LOAD      M0165D	// R_3rd ROT R START 1PLS
LOAD      M0165F	// R_3rd ROT R MOVE HOLD
AND NOT   M0165E	// R_3rd ROT R POS OK PLS
AND NOT   M0165C	// R_3rd ROT R HOLD CUT
OR LOAD
OUT       M0165F	// R_3rd ROT R MOVE HOLD
OUT       D002280.7	// R_3rd ROT R ABS POS MV
; L149
LOAD NOT  D002280.E	// R_3rd ROT R Stop Servo
TON       T0765 10	// R_3rd ROT R ºñ»óÁ¤Áö OFF
; L150
LOAD      M00600	// EMERGENCY ALARM
OR        M0215F	// T)R_3rd ROT R STOP
AND       T0765	// R_3rd ROT R ºñ»óÁ¤Áö OFF
OUT       D002280.E	// R_3rd ROT R Stop Servo
; L152
LOAD NOT  D001280.E	// R_2nd ROT R Limit +
AND NOT   D001280.F	// R_2nd ROT R Limit -
TON       T0915 2	// R_3rd ROT R LMT RST TM

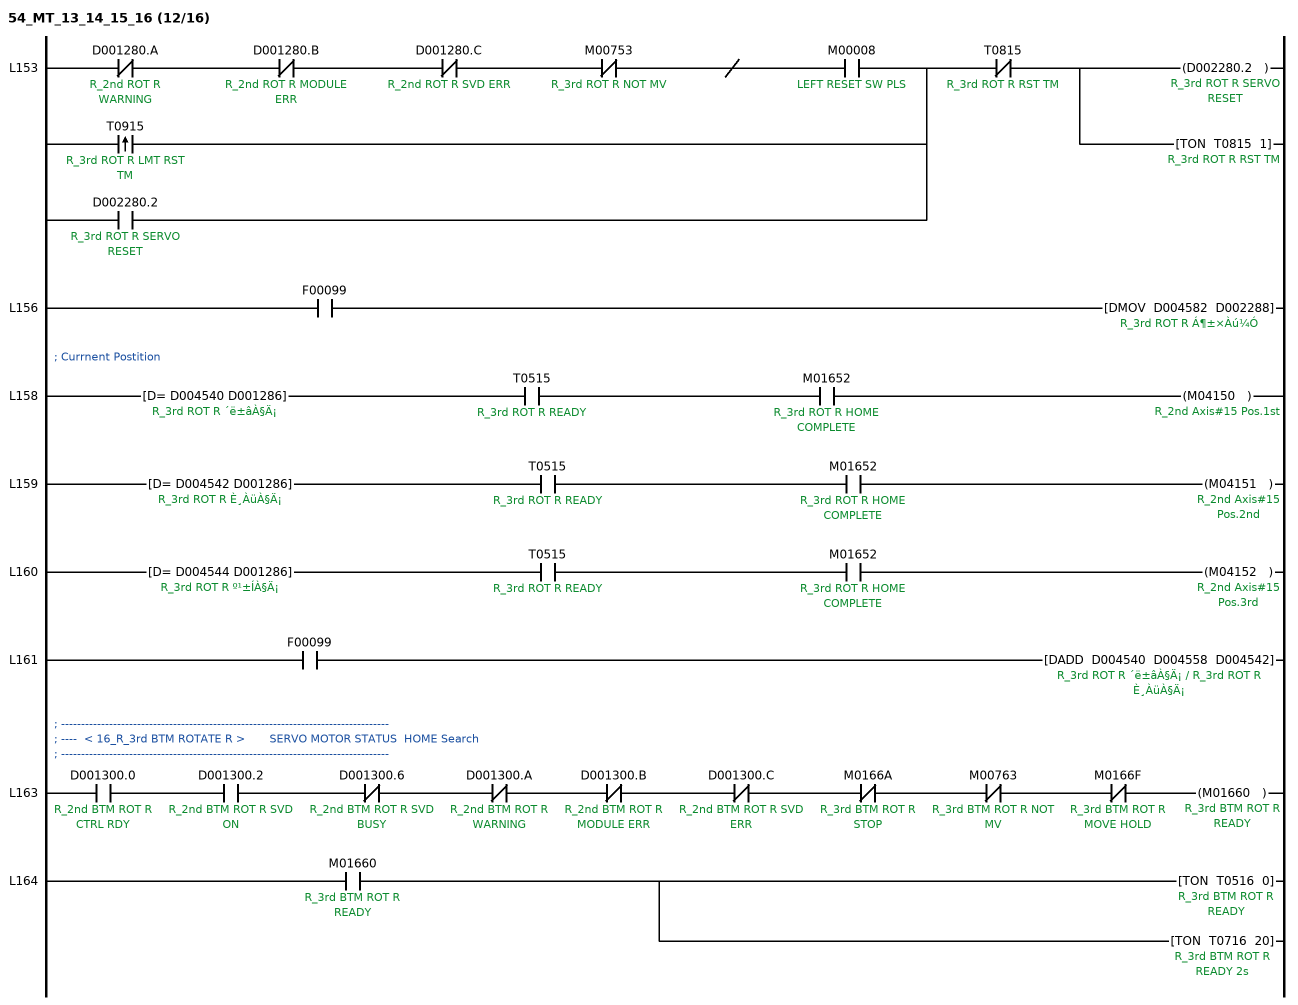
; L153
LOAD NOT  D001280.A	// R_2nd ROT R WARNING
AND NOT   D001280.B	// R_2nd ROT R MODULE ERR
AND NOT   D001280.C	// R_2nd ROT R SVD ERR
AND NOT   M00753	// R_3rd ROT R NOT MV
NOT
AND       M00008	// LEFT RESET SW PLS
ORP       T0915	// R_3rd ROT R LMT RST TM
OR        D002280.2	// R_3rd ROT R SERVO RESET
AND NOT   T0815	// R_3rd ROT R RST TM
OUT       D002280.2	// R_3rd ROT R SERVO RESET
TON       T0815 1	// R_3rd ROT R RST TM
; L156
LOAD      F00099
DMOV      D004582 D002288	// R_3rd ROT R Á¶±×Àú¼Ó
// Currnent Postition
; L158
LOADD=    D004540 D001286	// R_3rd ROT R ´ë±âÀ§Ä¡
AND       T0515	// R_3rd ROT R READY
AND       M01652	// R_3rd ROT R HOME COMPLETE
OUT       M04150	// R_2nd Axis#15 Pos.1st
; L159
LOADD=    D004542 D001286	// R_3rd ROT R È¸ÀüÀ§Ä¡
AND       T0515	// R_3rd ROT R READY
AND       M01652	// R_3rd ROT R HOME COMPLETE
OUT       M04151	// R_2nd Axis#15 Pos.2nd
; L160
LOADD=    D004544 D001286	// R_3rd ROT R º¹±ÍÀ§Ä¡
AND       T0515	// R_3rd ROT R READY
AND       M01652	// R_3rd ROT R HOME COMPLETE
OUT       M04152	// R_2nd Axis#15 Pos.3rd
; L161
LOAD      F00099
DADD      D004540 D004558 D004542	// R_3rd ROT R ´ë±âÀ§Ä¡ / R_3rd ROT R È¸ÀüÀ§Ä¡
// ----------------------------------------------------------------------------------
// 
// ----  < 16_R_3rd BTM ROTATE R >       SERVO MOTOR STATUS  HOME Search
// 
// ----------------------------------------------------------------------------------
; L163
LOAD      D001300.0	// R_2nd BTM ROT R CTRL RDY
AND       D001300.2	// R_2nd BTM ROT R SVD ON
AND NOT   D001300.6	// R_2nd BTM ROT R SVD BUSY
AND NOT   D001300.A	// R_2nd BTM ROT R WARNING
AND NOT   D001300.B	// R_2nd BTM ROT R MODULE ERR
AND NOT   D001300.C	// R_2nd BTM ROT R SVD ERR
AND NOT   M0166A	// R_3rd BTM ROT R STOP
AND NOT   M00763	// R_3rd BTM ROT R NOT MV
AND NOT   M0166F	// R_3rd BTM ROT R MOVE HOLD
OUT       M01660	// R_3rd BTM ROT R READY
; L164
LOAD      M01660	// R_3rd BTM ROT R READY
TON       T0516 0	// R_3rd BTM ROT R READY
TON       T0716 20	// R_3rd BTM ROT R READY 2s

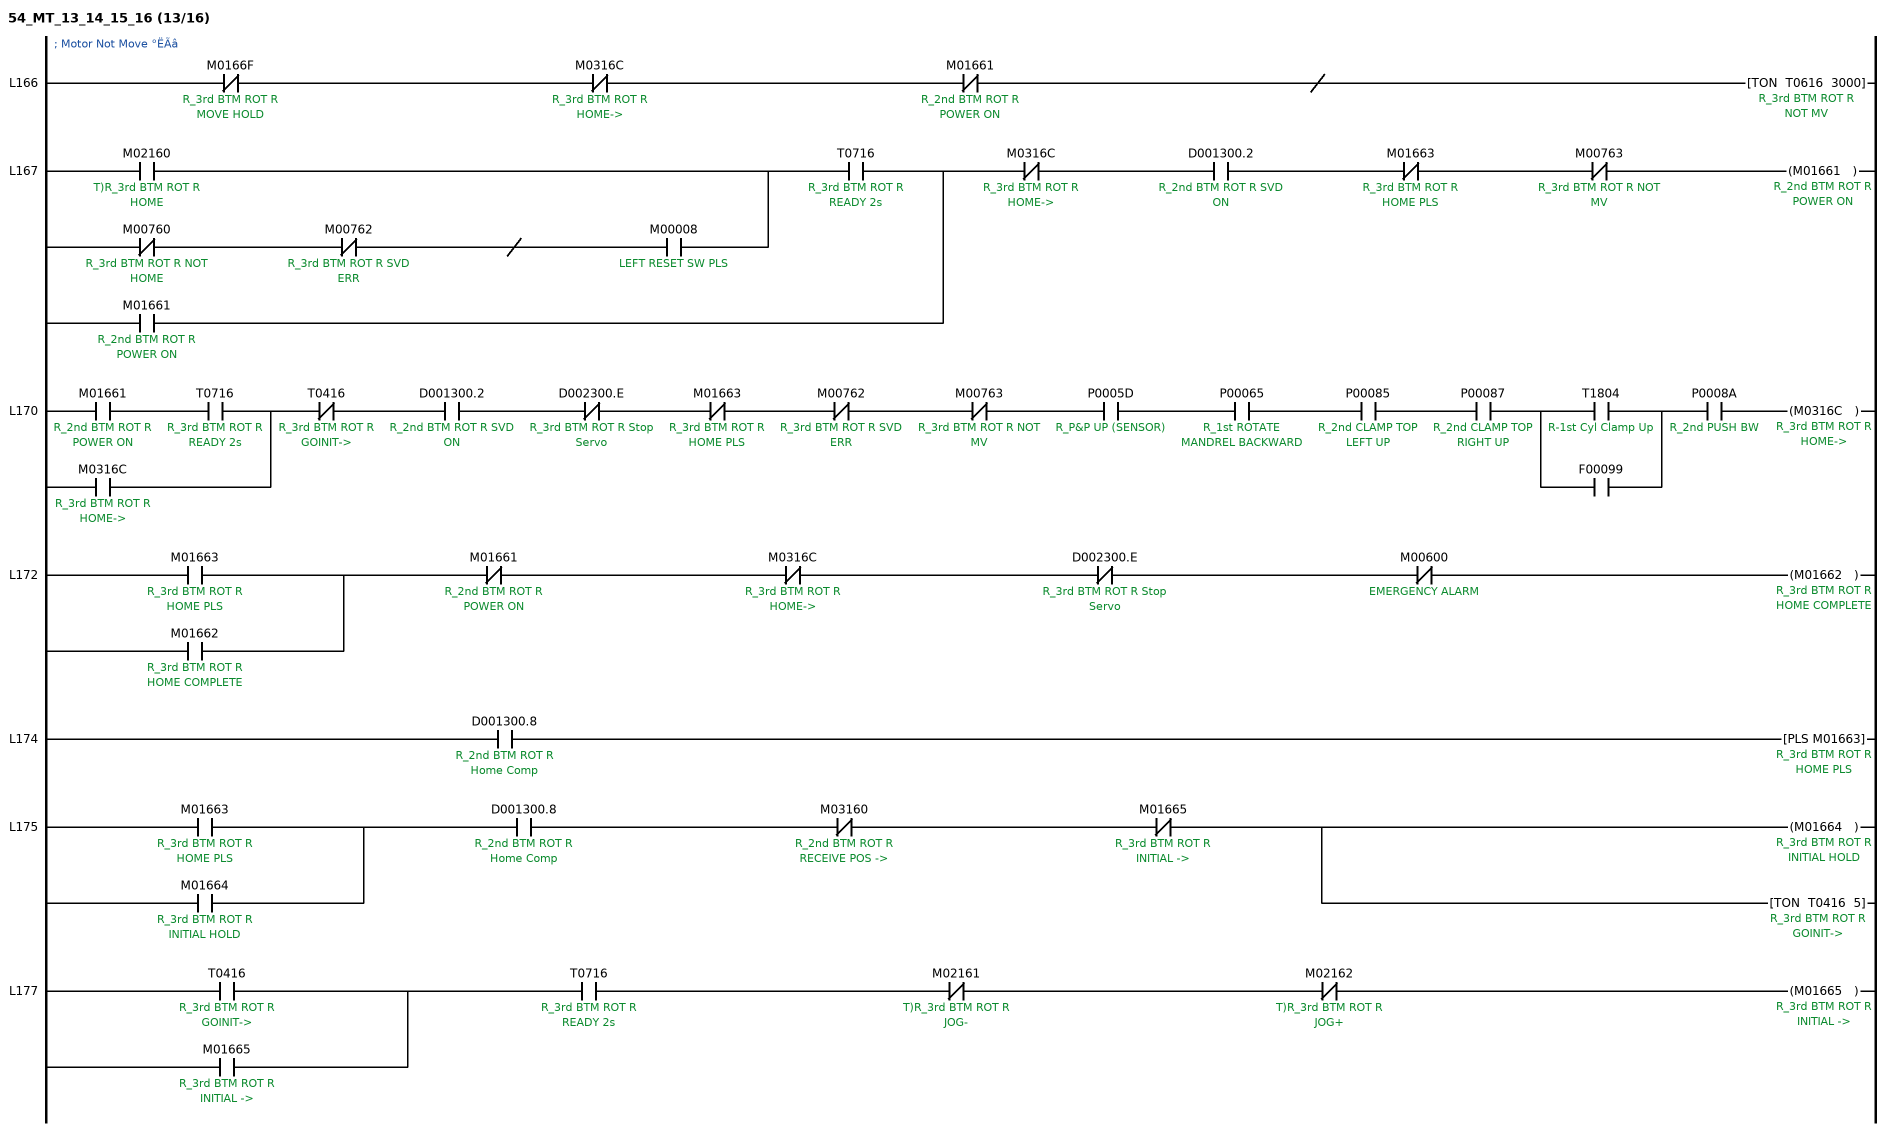
; L166
LOAD NOT  M0166F	// R_3rd BTM ROT R MOVE HOLD
AND NOT   M0316C	// R_3rd BTM ROT R HOME->
AND NOT   M01661	// R_2nd BTM ROT R POWER ON
NOT
TON       T0616 3000	// R_3rd BTM ROT R NOT MV
// output comment: Motor Not Move °ËÃâ
; L167
LOAD      M02160	// T)R_3rd BTM ROT R HOME
LOAD NOT  M00760	// R_3rd BTM ROT R NOT HOME
AND NOT   M00762	// R_3rd BTM ROT R SVD ERR
NOT
AND       M00008	// LEFT RESET SW PLS
OR LOAD
AND       T0716	// R_3rd BTM ROT R READY 2s
OR        M01661	// R_2nd BTM ROT R POWER ON
AND NOT   M0316C	// R_3rd BTM ROT R HOME->
AND       D001300.2	// R_2nd BTM ROT R SVD ON
AND NOT   M01663	// R_3rd BTM ROT R HOME PLS
AND NOT   M00763	// R_3rd BTM ROT R NOT MV
OUT       M01661	// R_2nd BTM ROT R POWER ON
; L170
LOAD      M01661	// R_2nd BTM ROT R POWER ON
AND       T0716	// R_3rd BTM ROT R READY 2s
OR        M0316C	// R_3rd BTM ROT R HOME->
AND NOT   T0416	// R_3rd BTM ROT R GOINIT->
AND       D001300.2	// R_2nd BTM ROT R SVD ON
AND NOT   D002300.E	// R_3rd BTM ROT R Stop Servo
AND NOT   M01663	// R_3rd BTM ROT R HOME PLS
AND NOT   M00762	// R_3rd BTM ROT R SVD ERR
AND NOT   M00763	// R_3rd BTM ROT R NOT MV
AND       P0005D	// R_P&P UP (SENSOR)
AND       P00065	// R_1st ROTATE MANDREL BACKWARD
AND       P00085	// R_2nd CLAMP TOP LEFT UP
AND       P00087	// R_2nd CLAMP TOP RIGHT UP
LOAD      T1804	// R-1st Cyl Clamp Up
OR        F00099
AND LOAD
AND       P0008A	// R_2nd PUSH BW
OUT       M0316C	// R_3rd BTM ROT R HOME->
; L172
LOAD      M01663	// R_3rd BTM ROT R HOME PLS
OR        M01662	// R_3rd BTM ROT R HOME COMPLETE
AND NOT   M01661	// R_2nd BTM ROT R POWER ON
AND NOT   M0316C	// R_3rd BTM ROT R HOME->
AND NOT   D002300.E	// R_3rd BTM ROT R Stop Servo
AND NOT   M00600	// EMERGENCY ALARM
OUT       M01662	// R_3rd BTM ROT R HOME COMPLETE
; L174
LOAD      D001300.8	// R_2nd BTM ROT R Home Comp 
OUTP      M01663	// R_3rd BTM ROT R HOME PLS
; L175
LOAD      M01663	// R_3rd BTM ROT R HOME PLS
OR        M01664	// R_3rd BTM ROT R INITIAL HOLD
AND       D001300.8	// R_2nd BTM ROT R Home Comp 
AND NOT   M03160	// R_2nd BTM ROT R RECEIVE POS ->
AND NOT   M01665	// R_3rd BTM ROT R INITIAL ->
OUT       M01664	// R_3rd BTM ROT R INITIAL HOLD
TON       T0416 5	// R_3rd BTM ROT R GOINIT->
; L177
LOAD      T0416	// R_3rd BTM ROT R GOINIT->
OR        M01665	// R_3rd BTM ROT R INITIAL ->
AND       T0716	// R_3rd BTM ROT R READY 2s
AND NOT   M02161	// T)R_3rd BTM ROT R JOG-
AND NOT   M02162	// T)R_3rd BTM ROT R JOG+
OUT       M01665	// R_3rd BTM ROT R INITIAL ->

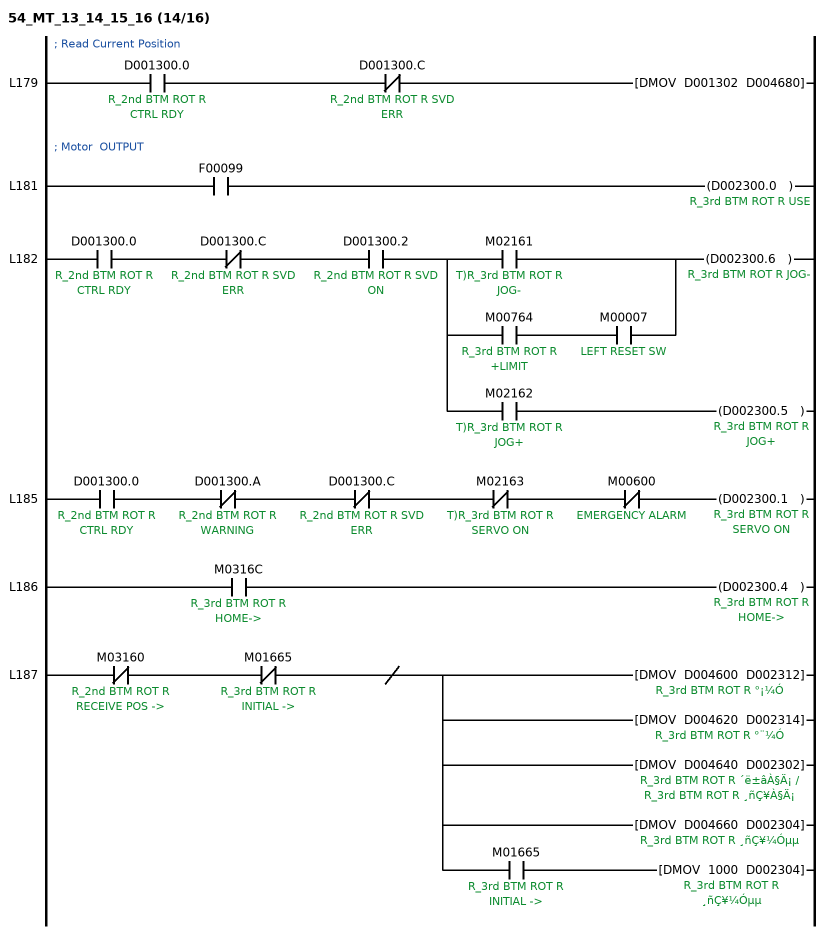
; L179
LOAD      D001300.0	// R_2nd BTM ROT R CTRL RDY
AND NOT   D001300.C	// R_2nd BTM ROT R SVD ERR
DMOV      D001302 D004680
// output comment: Read Current Position
//  Motor  OUTPUT
; L181
LOAD      F00099
OUT       D002300.0	// R_3rd BTM ROT R USE
; L182
LOAD      D001300.0	// R_2nd BTM ROT R CTRL RDY
AND NOT   D001300.C	// R_2nd BTM ROT R SVD ERR
AND       D001300.2	// R_2nd BTM ROT R SVD ON
MPUSH
LOAD      M02161	// T)R_3rd BTM ROT R JOG-
LOAD      M00764	// R_3rd BTM ROT R +LIMIT
AND       M00007	// LEFT RESET SW
OR LOAD
AND LOAD
OUT       D002300.6	// R_3rd BTM ROT R JOG-
MPOP
AND       M02162	// T)R_3rd BTM ROT R JOG+
OUT       D002300.5	// R_3rd BTM ROT R JOG+
; L185
LOAD      D001300.0	// R_2nd BTM ROT R CTRL RDY
AND NOT   D001300.A	// R_2nd BTM ROT R WARNING
AND NOT   D001300.C	// R_2nd BTM ROT R SVD ERR
AND NOT   M02163	// T)R_3rd BTM ROT R SERVO ON
AND NOT   M00600	// EMERGENCY ALARM
OUT       D002300.1	// R_3rd BTM ROT R SERVO ON
; L186
LOAD      M0316C	// R_3rd BTM ROT R HOME->
OUT       D002300.4	// R_3rd BTM ROT R HOME->
; L187
LOAD NOT  M03160	// R_2nd BTM ROT R RECEIVE POS ->
AND NOT   M01665	// R_3rd BTM ROT R INITIAL ->
NOT
DMOV      D004600 D002312	// R_3rd BTM ROT R °¡¼Ó
DMOV      D004620 D002314	// R_3rd BTM ROT R °¨¼Ó
DMOV      D004640 D002302	// R_3rd BTM ROT R ´ë±âÀ§Ä¡ / R_3rd BTM ROT R ¸ñÇ¥À§Ä¡
DMOV      D004660 D002304	// R_3rd BTM ROT R ¸ñÇ¥¼Óµµ
AND       M01665	// R_3rd BTM ROT R INITIAL ->
DMOV      1000 D002304	// R_3rd BTM ROT R ¸ñÇ¥¼Óµµ

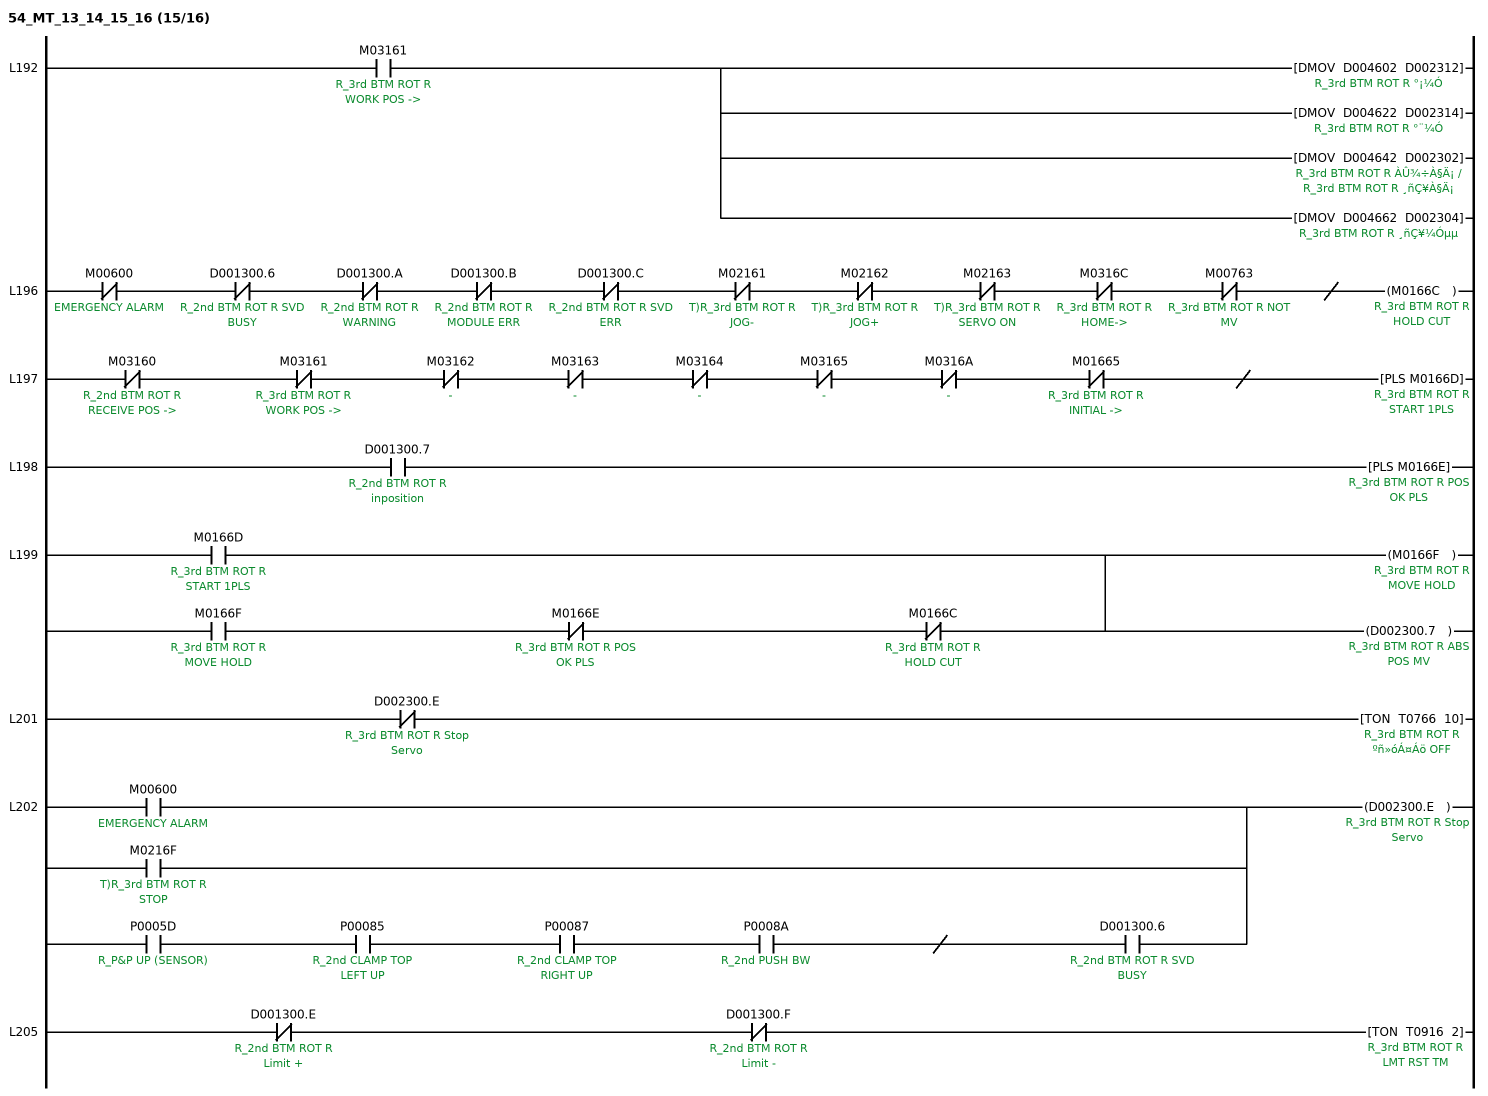
; L192
LOAD      M03161	// R_3rd BTM ROT R WORK POS ->
DMOV      D004602 D002312	// R_3rd BTM ROT R °¡¼Ó
DMOV      D004622 D002314	// R_3rd BTM ROT R °¨¼Ó
DMOV      D004642 D002302	// R_3rd BTM ROT R ÀÛ¾÷À§Ä¡ / R_3rd BTM ROT R ¸ñÇ¥À§Ä¡
DMOV      D004662 D002304	// R_3rd BTM ROT R ¸ñÇ¥¼Óµµ
; L196
LOAD NOT  M00600	// EMERGENCY ALARM
AND NOT   D001300.6	// R_2nd BTM ROT R SVD BUSY
AND NOT   D001300.A	// R_2nd BTM ROT R WARNING
AND NOT   D001300.B	// R_2nd BTM ROT R MODULE ERR
AND NOT   D001300.C	// R_2nd BTM ROT R SVD ERR
AND NOT   M02161	// T)R_3rd BTM ROT R JOG-
AND NOT   M02162	// T)R_3rd BTM ROT R JOG+
AND NOT   M02163	// T)R_3rd BTM ROT R SERVO ON
AND NOT   M0316C	// R_3rd BTM ROT R HOME->
AND NOT   M00763	// R_3rd BTM ROT R NOT MV
NOT
OUT       M0166C	// R_3rd BTM ROT R HOLD CUT
; L197
LOAD NOT  M03160	// R_2nd BTM ROT R RECEIVE POS ->
AND NOT   M03161	// R_3rd BTM ROT R WORK POS ->
AND NOT   M03162	// -
AND NOT   M03163	// -
AND NOT   M03164	// -
AND NOT   M03165	// -
AND NOT   M0316A	// -
AND NOT   M01665	// R_3rd BTM ROT R INITIAL ->
NOT
OUTP      M0166D	// R_3rd BTM ROT R START 1PLS
; L198
LOAD      D001300.7	// R_2nd BTM ROT R inposition
OUTP      M0166E	// R_3rd BTM ROT R POS OK PLS
; L199
LOAD      M0166D	// R_3rd BTM ROT R START 1PLS
LOAD      M0166F	// R_3rd BTM ROT R MOVE HOLD
AND NOT   M0166E	// R_3rd BTM ROT R POS OK PLS
AND NOT   M0166C	// R_3rd BTM ROT R HOLD CUT
OR LOAD
OUT       M0166F	// R_3rd BTM ROT R MOVE HOLD
OUT       D002300.7	// R_3rd BTM ROT R ABS POS MV
; L201
LOAD NOT  D002300.E	// R_3rd BTM ROT R Stop Servo
TON       T0766 10	// R_3rd BTM ROT R ºñ»óÁ¤Áö OFF
; L202
LOAD      M00600	// EMERGENCY ALARM
OR        M0216F	// T)R_3rd BTM ROT R STOP
LOAD      P0005D	// R_P&P UP (SENSOR)
AND       P00085	// R_2nd CLAMP TOP LEFT UP
AND       P00087	// R_2nd CLAMP TOP RIGHT UP
AND       P0008A	// R_2nd PUSH BW
NOT
AND       D001300.6	// R_2nd BTM ROT R SVD BUSY
OR LOAD
OUT       D002300.E	// R_3rd BTM ROT R Stop Servo
; L205
LOAD NOT  D001300.E	// R_2nd BTM ROT R Limit +
AND NOT   D001300.F	// R_2nd BTM ROT R Limit -
TON       T0916 2	// R_3rd BTM ROT R LMT RST TM

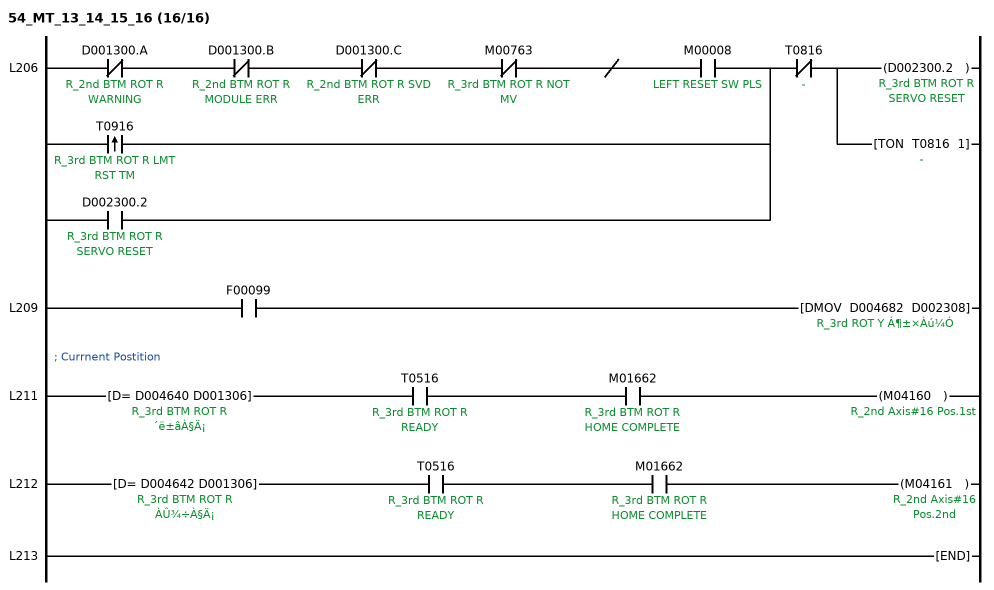
; L206
LOAD NOT  D001300.A	// R_2nd BTM ROT R WARNING
AND NOT   D001300.B	// R_2nd BTM ROT R MODULE ERR
AND NOT   D001300.C	// R_2nd BTM ROT R SVD ERR
AND NOT   M00763	// R_3rd BTM ROT R NOT MV
NOT
AND       M00008	// LEFT RESET SW PLS
ORP       T0916	// R_3rd BTM ROT R LMT RST TM
OR        D002300.2	// R_3rd BTM ROT R SERVO RESET
AND NOT   T0816	// -
OUT       D002300.2	// R_3rd BTM ROT R SERVO RESET
TON       T0816 1	// -
; L209
LOAD      F00099
DMOV      D004682 D002308	// R_3rd ROT Y Á¶±×Àú¼Ó
// Currnent Postition
; L211
LOADD=    D004640 D001306	// R_3rd BTM ROT R ´ë±âÀ§Ä¡
AND       T0516	// R_3rd BTM ROT R READY
AND       M01662	// R_3rd BTM ROT R HOME COMPLETE
OUT       M04160	// R_2nd Axis#16 Pos.1st
; L212
LOADD=    D004642 D001306	// R_3rd BTM ROT R ÀÛ¾÷À§Ä¡
AND       T0516	// R_3rd BTM ROT R READY
AND       M01662	// R_3rd BTM ROT R HOME COMPLETE
OUT       M04161	// R_2nd Axis#16 Pos.2nd
; L213
END

PROGRAM 55_MT_17_18_19_20 (task: ½ºÄµ ÇÁ·Î±×·¥)

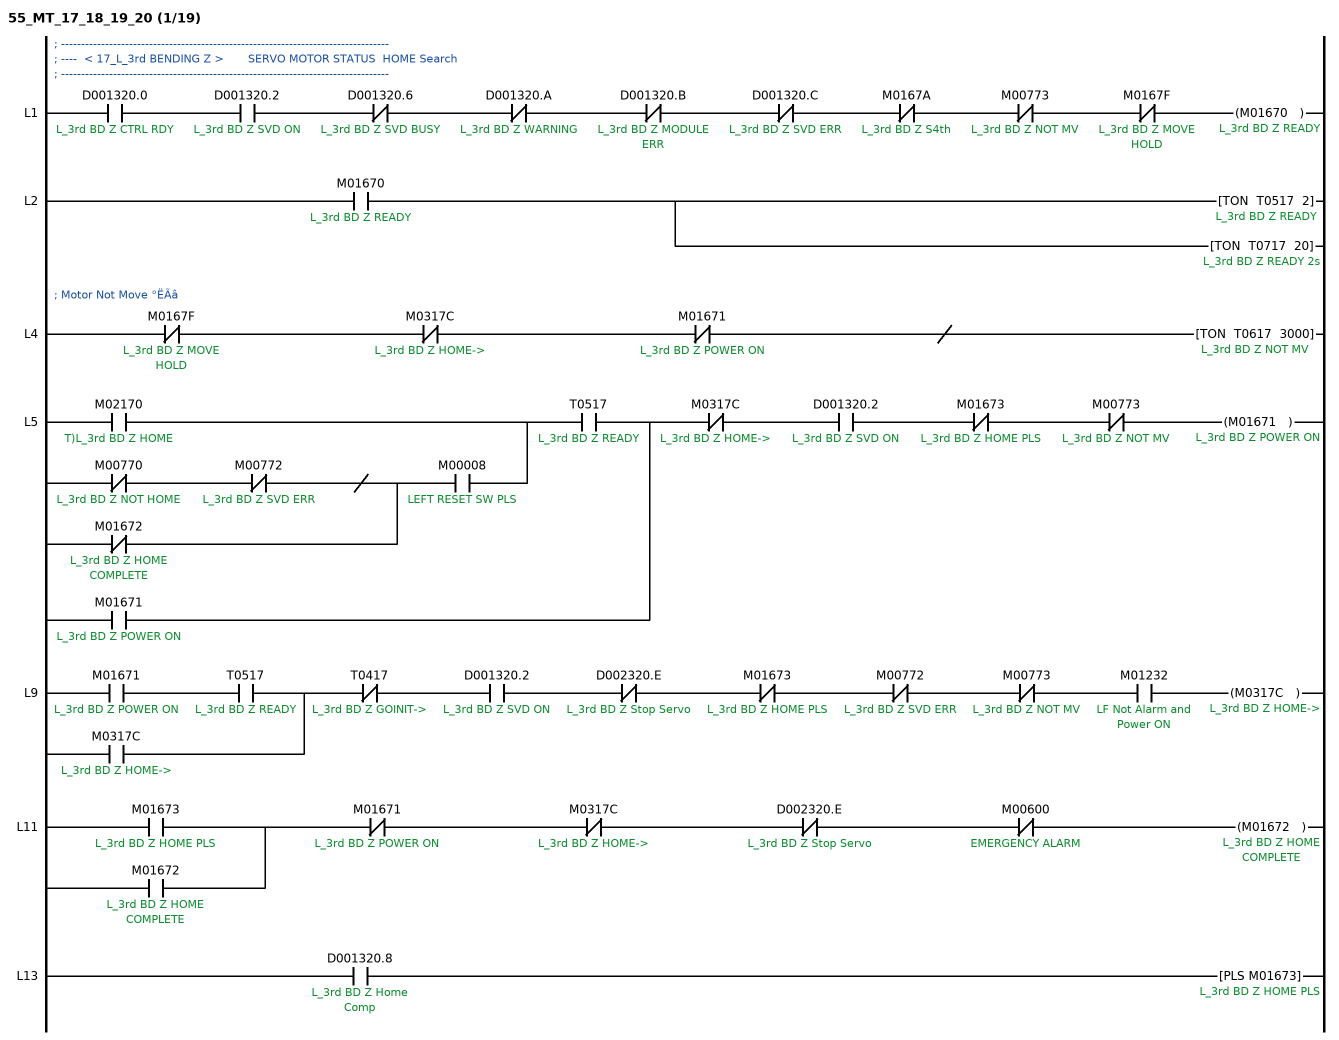
// ----------------------------------------------------------------------------------
// 
// ----  < 17_L_3rd BENDING Z >       SERVO MOTOR STATUS  HOME Search
// 
// ----------------------------------------------------------------------------------
; L1
LOAD      D001320.0	// L_3rd BD Z CTRL RDY
AND       D001320.2	// L_3rd BD Z SVD ON
AND NOT   D001320.6	// L_3rd BD Z SVD BUSY
AND NOT   D001320.A	// L_3rd BD Z WARNING
AND NOT   D001320.B	// L_3rd BD Z MODULE ERR
AND NOT   D001320.C	// L_3rd BD Z SVD ERR
AND NOT   M0167A	// L_3rd BD Z S4th
AND NOT   M00773	// L_3rd BD Z NOT MV
AND NOT   M0167F	// L_3rd BD Z MOVE HOLD
OUT       M01670	// L_3rd BD Z READY
; L2
LOAD      M01670	// L_3rd BD Z READY
TON       T0517 2	// L_3rd BD Z READY
TON       T0717 20	// L_3rd BD Z READY 2s
; L4
LOAD NOT  M0167F	// L_3rd BD Z MOVE HOLD
AND NOT   M0317C	// L_3rd BD Z HOME->
AND NOT   M01671	// L_3rd BD Z POWER ON
NOT
TON       T0617 3000	// L_3rd BD Z NOT MV
// output comment: Motor Not Move °ËÃâ
; L5
LOAD      M02170	// T)L_3rd BD Z HOME
LOAD NOT  M00770	// L_3rd BD Z NOT HOME
AND NOT   M00772	// L_3rd BD Z SVD ERR
NOT
OR NOT    M01672	// L_3rd BD Z HOME COMPLETE
AND       M00008	// LEFT RESET SW PLS
OR LOAD
AND       T0517	// L_3rd BD Z READY
OR        M01671	// L_3rd BD Z POWER ON
AND NOT   M0317C	// L_3rd BD Z HOME->
AND       D001320.2	// L_3rd BD Z SVD ON
AND NOT   M01673	// L_3rd BD Z HOME PLS
AND NOT   M00773	// L_3rd BD Z NOT MV
OUT       M01671	// L_3rd BD Z POWER ON
; L9
LOAD      M01671	// L_3rd BD Z POWER ON
AND       T0517	// L_3rd BD Z READY
OR        M0317C	// L_3rd BD Z HOME->
AND NOT   T0417	// L_3rd BD Z GOINIT->
AND       D001320.2	// L_3rd BD Z SVD ON
AND NOT   D002320.E	// L_3rd BD Z Stop Servo
AND NOT   M01673	// L_3rd BD Z HOME PLS
AND NOT   M00772	// L_3rd BD Z SVD ERR
AND NOT   M00773	// L_3rd BD Z NOT MV
AND       M01232	// LF Not Alarm and Power ON
OUT       M0317C	// L_3rd BD Z HOME->
; L11
LOAD      M01673	// L_3rd BD Z HOME PLS
OR        M01672	// L_3rd BD Z HOME COMPLETE
AND NOT   M01671	// L_3rd BD Z POWER ON
AND NOT   M0317C	// L_3rd BD Z HOME->
AND NOT   D002320.E	// L_3rd BD Z Stop Servo
AND NOT   M00600	// EMERGENCY ALARM
OUT       M01672	// L_3rd BD Z HOME COMPLETE
; L13
LOAD      D001320.8	// L_3rd BD Z Home Comp
OUTP      M01673	// L_3rd BD Z HOME PLS

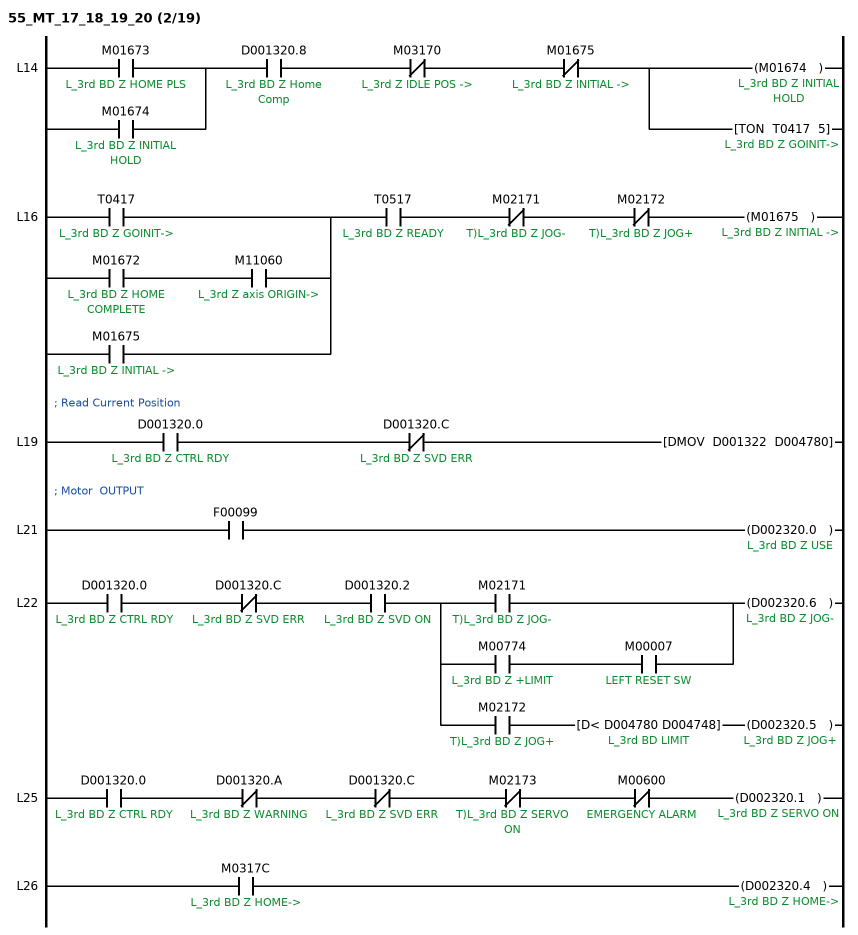
; L14
LOAD      M01673	// L_3rd BD Z HOME PLS
OR        M01674	// L_3rd BD Z INITIAL HOLD
AND       D001320.8	// L_3rd BD Z Home Comp
AND NOT   M03170	// L_3rd Z IDLE POS ->
AND NOT   M01675	// L_3rd BD Z INITIAL ->
OUT       M01674	// L_3rd BD Z INITIAL HOLD
TON       T0417 5	// L_3rd BD Z GOINIT->
; L16
LOAD      T0417	// L_3rd BD Z GOINIT->
LOAD      M01672	// L_3rd BD Z HOME COMPLETE
AND       M11060	// L_3rd Z axis ORIGIN->
OR LOAD
OR        M01675	// L_3rd BD Z INITIAL ->
AND       T0517	// L_3rd BD Z READY
AND NOT   M02171	// T)L_3rd BD Z JOG-
AND NOT   M02172	// T)L_3rd BD Z JOG+
OUT       M01675	// L_3rd BD Z INITIAL ->
; L19
LOAD      D001320.0	// L_3rd BD Z CTRL RDY
AND NOT   D001320.C	// L_3rd BD Z SVD ERR
DMOV      D001322 D004780
// output comment: Read Current Position
//  Motor  OUTPUT
; L21
LOAD      F00099
OUT       D002320.0	// L_3rd BD Z USE
; L22
LOAD      D001320.0	// L_3rd BD Z CTRL RDY
AND NOT   D001320.C	// L_3rd BD Z SVD ERR
AND       D001320.2	// L_3rd BD Z SVD ON
MPUSH
LOAD      M02171	// T)L_3rd BD Z JOG-
LOAD      M00774	// L_3rd BD Z +LIMIT
AND       M00007	// LEFT RESET SW
OR LOAD
AND LOAD
OUT       D002320.6	// L_3rd BD Z JOG-
MPOP
AND       M02172	// T)L_3rd BD Z JOG+
ANDD<     D004780 D004748	// L_3rd BD LIMIT
OUT       D002320.5	// L_3rd BD Z JOG+
; L25
LOAD      D001320.0	// L_3rd BD Z CTRL RDY
AND NOT   D001320.A	// L_3rd BD Z WARNING
AND NOT   D001320.C	// L_3rd BD Z SVD ERR
AND NOT   M02173	// T)L_3rd BD Z SERVO ON
AND NOT   M00600	// EMERGENCY ALARM
OUT       D002320.1	// L_3rd BD Z SERVO ON
; L26
LOAD      M0317C	// L_3rd BD Z HOME->
OUT       D002320.4	// L_3rd BD Z HOME->

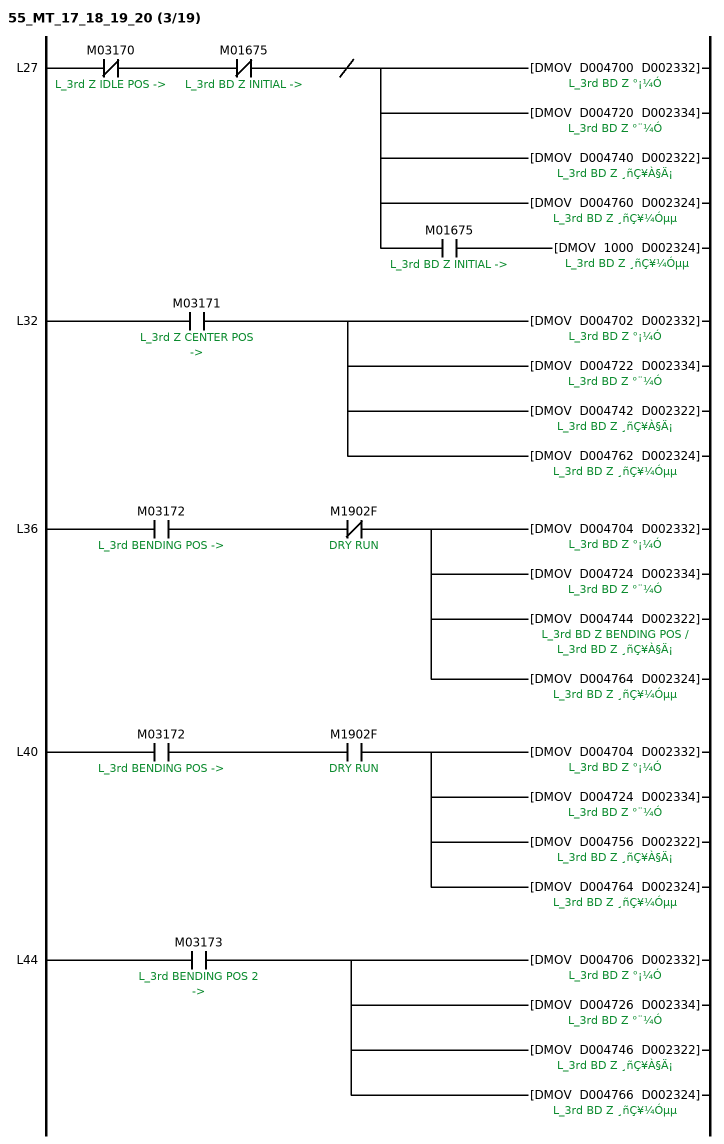
; L27
LOAD NOT  M03170	// L_3rd Z IDLE POS ->
AND NOT   M01675	// L_3rd BD Z INITIAL ->
NOT
DMOV      D004700 D002332	// L_3rd BD Z °¡¼Ó
DMOV      D004720 D002334	// L_3rd BD Z °¨¼Ó
DMOV      D004740 D002322	// L_3rd BD Z ¸ñÇ¥À§Ä¡
DMOV      D004760 D002324	// L_3rd BD Z ¸ñÇ¥¼Óµµ
AND       M01675	// L_3rd BD Z INITIAL ->
DMOV      1000 D002324	// L_3rd BD Z ¸ñÇ¥¼Óµµ
; L32
LOAD      M03171	// L_3rd Z CENTER POS ->
DMOV      D004702 D002332	// L_3rd BD Z °¡¼Ó
DMOV      D004722 D002334	// L_3rd BD Z °¨¼Ó
DMOV      D004742 D002322	// L_3rd BD Z ¸ñÇ¥À§Ä¡
DMOV      D004762 D002324	// L_3rd BD Z ¸ñÇ¥¼Óµµ
; L36
LOAD      M03172	// L_3rd BENDING POS ->
AND NOT   M1902F	// DRY RUN
DMOV      D004704 D002332	// L_3rd BD Z °¡¼Ó
DMOV      D004724 D002334	// L_3rd BD Z °¨¼Ó
DMOV      D004744 D002322	// L_3rd BD Z BENDING POS / L_3rd BD Z ¸ñÇ¥À§Ä¡
DMOV      D004764 D002324	// L_3rd BD Z ¸ñÇ¥¼Óµµ
; L40
LOAD      M03172	// L_3rd BENDING POS ->
AND       M1902F	// DRY RUN
DMOV      D004704 D002332	// L_3rd BD Z °¡¼Ó
DMOV      D004724 D002334	// L_3rd BD Z °¨¼Ó
DMOV      D004756 D002322	// L_3rd BD Z ¸ñÇ¥À§Ä¡
DMOV      D004764 D002324	// L_3rd BD Z ¸ñÇ¥¼Óµµ
; L44
LOAD      M03173	// L_3rd BENDING POS 2 ->
DMOV      D004706 D002332	// L_3rd BD Z °¡¼Ó
DMOV      D004726 D002334	// L_3rd BD Z °¨¼Ó
DMOV      D004746 D002322	// L_3rd BD Z ¸ñÇ¥À§Ä¡
DMOV      D004766 D002324	// L_3rd BD Z ¸ñÇ¥¼Óµµ

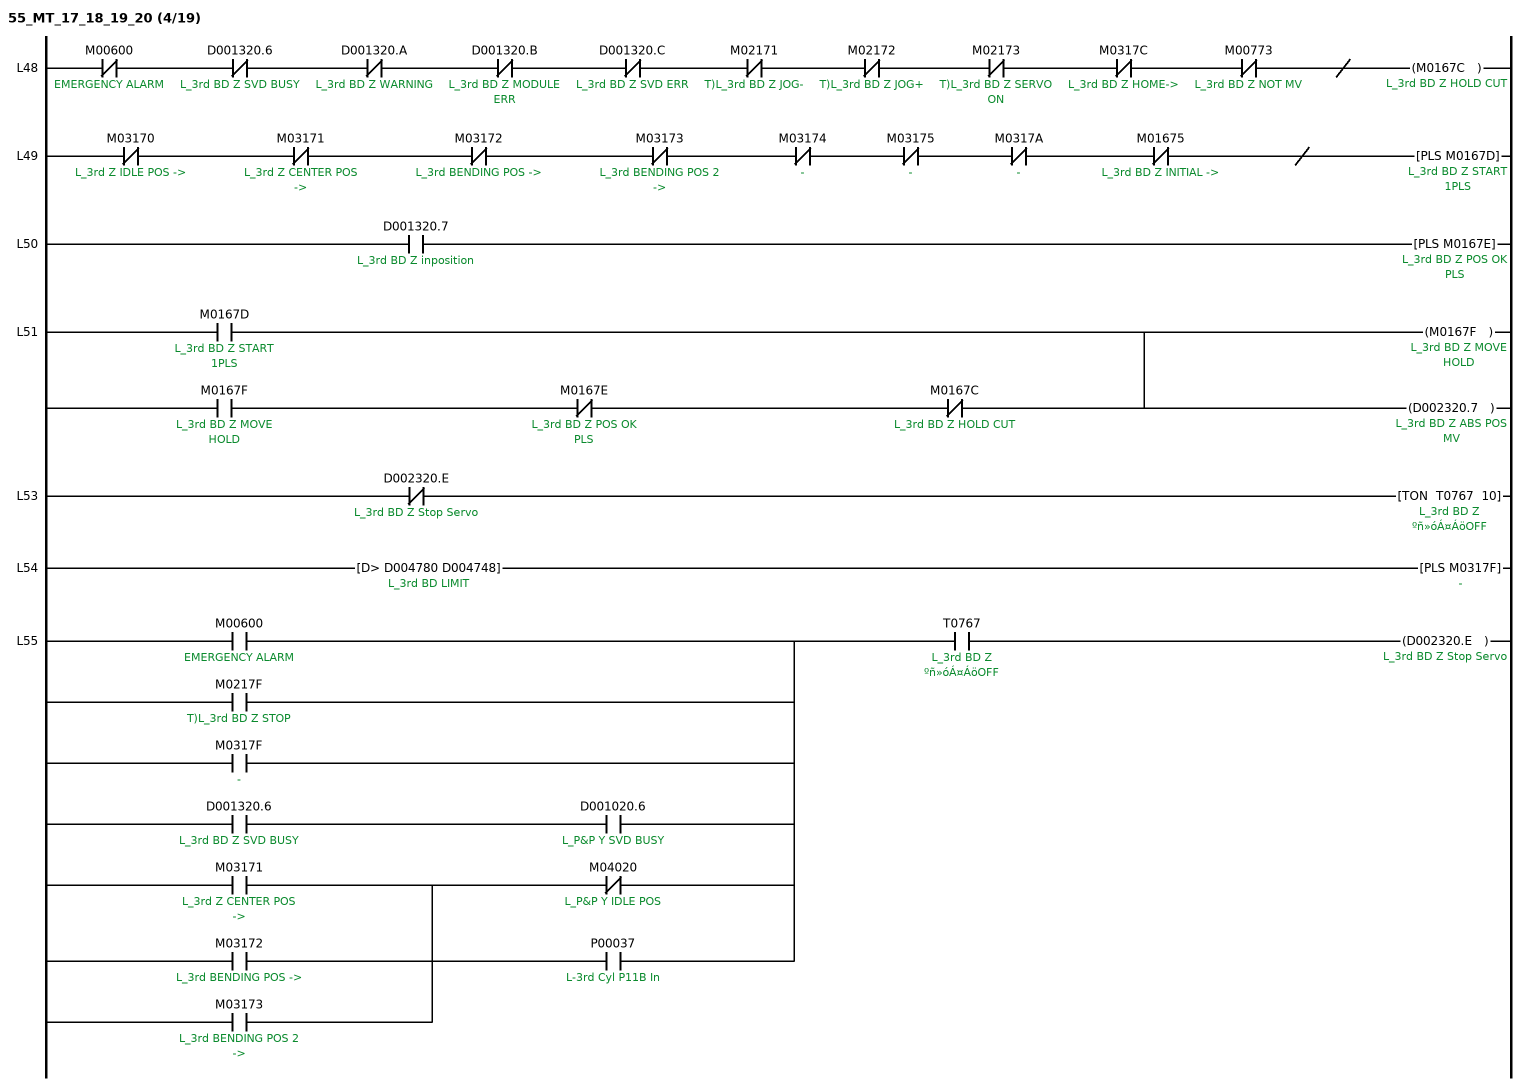
; L48
LOAD NOT  M00600	// EMERGENCY ALARM
AND NOT   D001320.6	// L_3rd BD Z SVD BUSY
AND NOT   D001320.A	// L_3rd BD Z WARNING
AND NOT   D001320.B	// L_3rd BD Z MODULE ERR
AND NOT   D001320.C	// L_3rd BD Z SVD ERR
AND NOT   M02171	// T)L_3rd BD Z JOG-
AND NOT   M02172	// T)L_3rd BD Z JOG+
AND NOT   M02173	// T)L_3rd BD Z SERVO ON
AND NOT   M0317C	// L_3rd BD Z HOME->
AND NOT   M00773	// L_3rd BD Z NOT MV
NOT
OUT       M0167C	// L_3rd BD Z HOLD CUT
; L49
LOAD NOT  M03170	// L_3rd Z IDLE POS ->
AND NOT   M03171	// L_3rd Z CENTER POS ->
AND NOT   M03172	// L_3rd BENDING POS ->
AND NOT   M03173	// L_3rd BENDING POS 2 ->
AND NOT   M03174	// -
AND NOT   M03175	// -
AND NOT   M0317A	// -
AND NOT   M01675	// L_3rd BD Z INITIAL ->
NOT
OUTP      M0167D	// L_3rd BD Z START 1PLS
; L50
LOAD      D001320.7	// L_3rd BD Z inposition
OUTP      M0167E	// L_3rd BD Z POS OK PLS
; L51
LOAD      M0167D	// L_3rd BD Z START 1PLS
LOAD      M0167F	// L_3rd BD Z MOVE HOLD
AND NOT   M0167E	// L_3rd BD Z POS OK PLS
AND NOT   M0167C	// L_3rd BD Z HOLD CUT
OR LOAD
OUT       M0167F	// L_3rd BD Z MOVE HOLD
OUT       D002320.7	// L_3rd BD Z ABS POS MV
; L53
LOAD NOT  D002320.E	// L_3rd BD Z Stop Servo
TON       T0767 10	// L_3rd BD Z ºñ»óÁ¤ÁöOFF
; L54
LOADD>    D004780 D004748	// L_3rd BD LIMIT
OUTP      M0317F	// -
; L55
LOAD      M00600	// EMERGENCY ALARM
OR        M0217F	// T)L_3rd BD Z STOP
OR        M0317F	// -
LOAD      D001320.6	// L_3rd BD Z SVD BUSY
AND       D001020.6	// L_P&P Y SVD BUSY
OR LOAD
LOAD      M03171	// L_3rd Z CENTER POS ->
OR        M03172	// L_3rd BENDING POS ->
OR        M03173	// L_3rd BENDING POS 2 ->
LOAD NOT  M04020	// L_P&P Y IDLE POS
OR        P00037	// L-3rd Cyl P11B In
AND LOAD
OR LOAD
AND       T0767	// L_3rd BD Z ºñ»óÁ¤ÁöOFF
OUT       D002320.E	// L_3rd BD Z Stop Servo

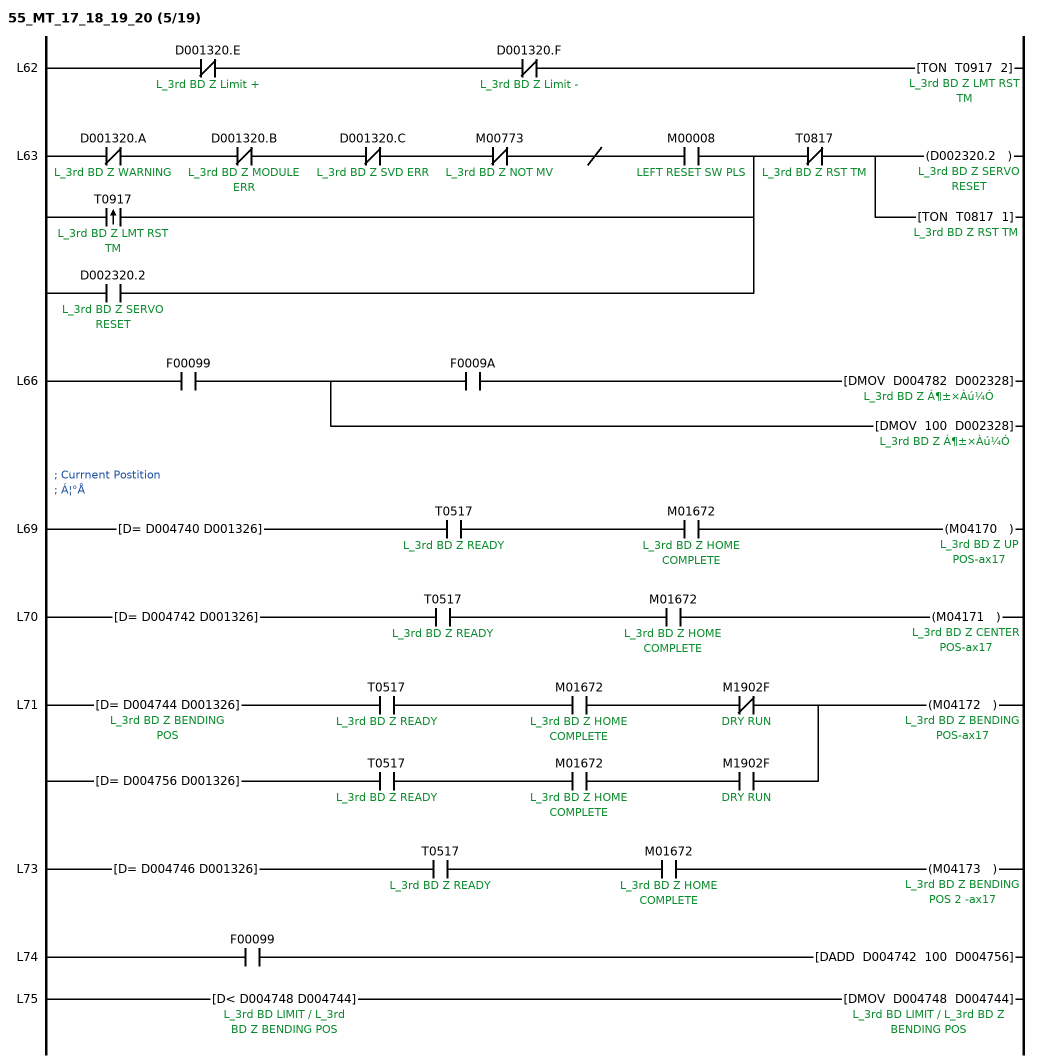
; L62
LOAD NOT  D001320.E	// L_3rd BD Z Limit +
AND NOT   D001320.F	// L_3rd BD Z Limit -
TON       T0917 2	// L_3rd BD Z LMT RST TM
; L63
LOAD NOT  D001320.A	// L_3rd BD Z WARNING
AND NOT   D001320.B	// L_3rd BD Z MODULE ERR
AND NOT   D001320.C	// L_3rd BD Z SVD ERR
AND NOT   M00773	// L_3rd BD Z NOT MV
NOT
AND       M00008	// LEFT RESET SW PLS
ORP       T0917	// L_3rd BD Z LMT RST TM
OR        D002320.2	// L_3rd BD Z SERVO RESET
AND NOT   T0817	// L_3rd BD Z RST TM
OUT       D002320.2	// L_3rd BD Z SERVO RESET
TON       T0817 1	// L_3rd BD Z RST TM
; L66
LOAD      F00099
MPUSH
AND       F0009A
DMOV      D004782 D002328	// L_3rd BD Z Á¶±×Àú¼Ó
MPOP
DMOV      100 D002328	// L_3rd BD Z Á¶±×Àú¼Ó
// Currnent Postition
; L69
LOADD=    D004740 D001326
AND       T0517	// L_3rd BD Z READY
AND       M01672	// L_3rd BD Z HOME COMPLETE
OUT       M04170	// L_3rd BD Z UP POS-ax17
// output comment: Á¦°Å
; L70
LOADD=    D004742 D001326
AND       T0517	// L_3rd BD Z READY
AND       M01672	// L_3rd BD Z HOME COMPLETE
OUT       M04171	// L_3rd BD Z CENTER POS-ax17
; L71
LOADD=    D004744 D001326	// L_3rd BD Z BENDING POS
AND       T0517	// L_3rd BD Z READY
AND       M01672	// L_3rd BD Z HOME COMPLETE
AND NOT   M1902F	// DRY RUN
LOADD=    D004756 D001326
AND       T0517	// L_3rd BD Z READY
AND       M01672	// L_3rd BD Z HOME COMPLETE
AND       M1902F	// DRY RUN
OR LOAD
OUT       M04172	// L_3rd BD Z BENDING POS-ax17
; L73
LOADD=    D004746 D001326
AND       T0517	// L_3rd BD Z READY
AND       M01672	// L_3rd BD Z HOME COMPLETE
OUT       M04173	// L_3rd BD Z BENDING POS 2 -ax17
; L74
LOAD      F00099
DADD      D004742 100 D004756
; L75
LOADD<    D004748 D004744	// L_3rd BD LIMIT / L_3rd BD Z BENDING POS
DMOV      D004748 D004744	// L_3rd BD LIMIT / L_3rd BD Z BENDING POS

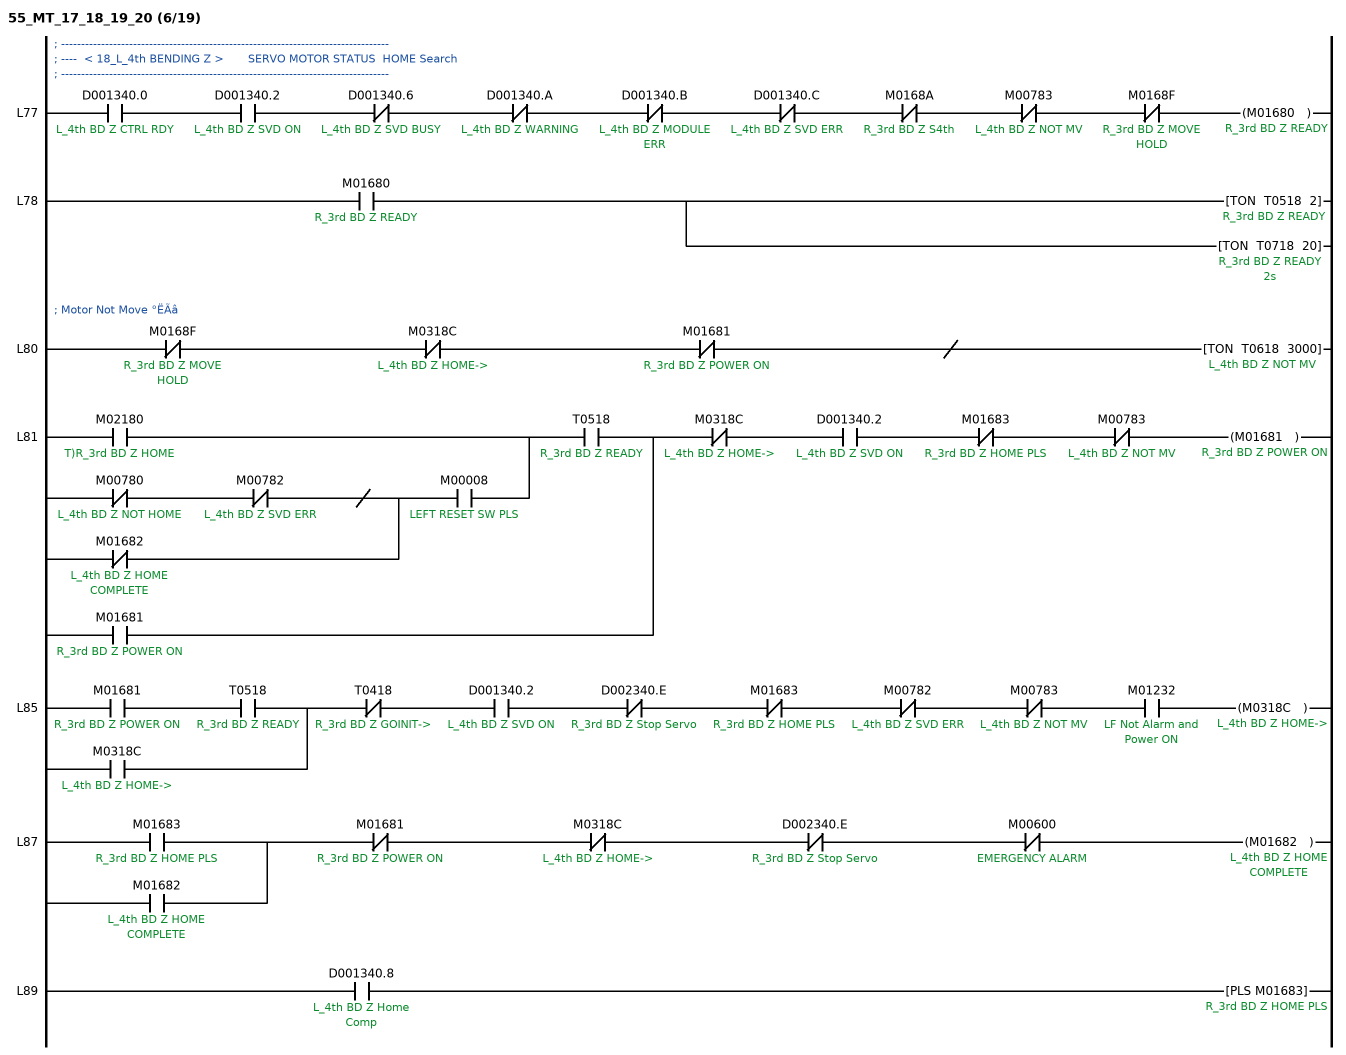
// ----------------------------------------------------------------------------------
// 
// ----  < 18_L_4th BENDING Z >       SERVO MOTOR STATUS  HOME Search
// 
// ----------------------------------------------------------------------------------
; L77
LOAD      D001340.0	// L_4th BD Z CTRL RDY
AND       D001340.2	// L_4th BD Z SVD ON
AND NOT   D001340.6	// L_4th BD Z SVD BUSY
AND NOT   D001340.A	// L_4th BD Z WARNING
AND NOT   D001340.B	// L_4th BD Z MODULE ERR
AND NOT   D001340.C	// L_4th BD Z SVD ERR
AND NOT   M0168A	// R_3rd BD Z S4th
AND NOT   M00783	// L_4th BD Z NOT MV
AND NOT   M0168F	// R_3rd BD Z MOVE HOLD
OUT       M01680	// R_3rd BD Z READY
; L78
LOAD      M01680	// R_3rd BD Z READY
TON       T0518 2	// R_3rd BD Z READY
TON       T0718 20	// R_3rd BD Z READY 2s
; L80
LOAD NOT  M0168F	// R_3rd BD Z MOVE HOLD
AND NOT   M0318C	// L_4th BD Z HOME->
AND NOT   M01681	// R_3rd BD Z POWER ON
NOT
TON       T0618 3000	// L_4th BD Z NOT MV
// output comment: Motor Not Move °ËÃâ
; L81
LOAD      M02180	// T)R_3rd BD Z HOME
LOAD NOT  M00780	// L_4th BD Z NOT HOME
AND NOT   M00782	// L_4th BD Z SVD ERR
NOT
OR NOT    M01682	// L_4th BD Z HOME COMPLETE
AND       M00008	// LEFT RESET SW PLS
OR LOAD
AND       T0518	// R_3rd BD Z READY
OR        M01681	// R_3rd BD Z POWER ON
AND NOT   M0318C	// L_4th BD Z HOME->
AND       D001340.2	// L_4th BD Z SVD ON
AND NOT   M01683	// R_3rd BD Z HOME PLS
AND NOT   M00783	// L_4th BD Z NOT MV
OUT       M01681	// R_3rd BD Z POWER ON
; L85
LOAD      M01681	// R_3rd BD Z POWER ON
AND       T0518	// R_3rd BD Z READY
OR        M0318C	// L_4th BD Z HOME->
AND NOT   T0418	// R_3rd BD Z GOINIT->
AND       D001340.2	// L_4th BD Z SVD ON
AND NOT   D002340.E	// R_3rd BD Z Stop Servo
AND NOT   M01683	// R_3rd BD Z HOME PLS
AND NOT   M00782	// L_4th BD Z SVD ERR
AND NOT   M00783	// L_4th BD Z NOT MV
AND       M01232	// LF Not Alarm and Power ON
OUT       M0318C	// L_4th BD Z HOME->
; L87
LOAD      M01683	// R_3rd BD Z HOME PLS
OR        M01682	// L_4th BD Z HOME COMPLETE
AND NOT   M01681	// R_3rd BD Z POWER ON
AND NOT   M0318C	// L_4th BD Z HOME->
AND NOT   D002340.E	// R_3rd BD Z Stop Servo
AND NOT   M00600	// EMERGENCY ALARM
OUT       M01682	// L_4th BD Z HOME COMPLETE
; L89
LOAD      D001340.8	// L_4th BD Z Home Comp
OUTP      M01683	// R_3rd BD Z HOME PLS

